LIN {X 0,Y 506.276,Z 611.91,A -85,B 0,C 180,E1 5620.333,E2 5620.333} C_VEL
LIN {X 0,Y 503.8,Z 611.91,A -85,B 0,C 180,E1 5621.794,E2 5621.794} C_VEL
LIN {X 0,Y 498.576,Z 611.91,A -85,B 0,C 180,E1 5623.986,E2 5623.986} C_VEL
LIN {X 0,Y 498.505,Z 611.91,A -85,B 0,C 180,E1 5624.239,E2 5624.239} C_VEL
LIN {X 0,Y 498.52,Z 611.91,A -85,B 0,C 180,E1 5630.373,E2 5630.373} C_VEL
LIN {X 0,Y 498.56,Z 611.91,A -85,B 0,C 180,E1 5636.864,E2 5636.864} C_VEL
LIN {X 0,Y 498.673,Z 612.016,A -85,B 0,C 180,E1 5638.544,E2 5638.544} C_VEL
LIN {X 0,Y 512.313,Z 645.051,A -85,B 0,C 180,E1 5639.998,E2 5639.998} C_VEL
LIN {X 0,Y 510.936,Z 684.615,A -85,B 0,C 180,E1 5640.995,E2 5640.995} C_VEL
LIN {X 0,Y 508.94,Z 720.292,A -85,B 0,C 180,E1 5642.602,E2 5642.602} C_VEL
LIN {X 0,Y 506.706,Z 753.658,A -85,B 0,C 180,E1 5644.799,E2 5644.799} C_VEL
LIN {X 0,Y 504.225,Z 785.399,A -85,B 0,C 180,E1 5647.723,E2 5647.723} C_VEL
LIN {X 0,Y 502.28,Z 810.959,A -85,B 0,C 180,E1 5650.895,E2 5650.895} C_VEL
LIN {X 0,Y 500.766,Z 834.651,A -85,B 0,C 180,E1 5654.902,E2 5654.902} C_VEL
LIN {X 0,Y 499.92,Z 850.471,A -85,B 0,C 180,E1 5658.647,E2 5658.647} C_VEL
LIN {X 0,Y 499.661,Z 861.793,A -85,B 0,C 180,E1 5662.601,E2 5662.601} C_VEL
LIN {X 0,Y 499.493,Z 868.21,A -85,B 0,C 180,E1 5666.524,E2 5666.524} C_VEL
LIN {X 0,Y 499.463,Z 870,A -85,B 0,C 180,E1 5670,E2 5670} C_VEL
LIN {X 0,Y 499.553,Z 867.136,A -85,B 0,C 180,E1 5674.346,E2 5674.346} C_VEL
LIN {X 0,Y 499.754,Z 858.648,A -85,B 0,C 180,E1 5678.713,E2 5678.713} C_VEL
LIN {X 0,Y 500.276,Z 843.684,A -85,B 0,C 180,E1 5683.12,E2 5683.12} C_VEL
LIN {X 0,Y 501.297,Z 824.914,A -85,B 0,C 180,E1 5686.9,E2 5686.9} C_VEL
LIN {X 0,Y 503.025,Z 800.805,A -85,B 0,C 180,E1 5690.481,E2 5690.481} C_VEL
LIN {X 0,Y 505.254,Z 771.947,A -85,B 0,C 180,E1 5693.626,E2 5693.626} C_VEL
LIN {X 0,Y 507.724,Z 739.674,A -85,B 0,C 180,E1 5696.213,E2 5696.213} C_VEL
LIN {X 0,Y 510.037,Z 703.559,A -85,B 0,C 180,E1 5698.236,E2 5698.236} C_VEL
LIN {X 0,Y 511.594,Z 668.352,A -85,B 0,C 180,E1 5699.506,E2 5699.506} C_VEL
LIN {X 0,Y 511.782,Z 643.626,A -85,B 0,C 180,E1 5700.064,E2 5700.064} C_VEL
LIN {X 0,Y 498.658,Z 611.91,A -85,B 0,C 180,E1 5701.494,E2 5701.494} C_VEL
LIN {X 0,Y 498.497,Z 611.91,A -85,B 0,C 180,E1 5707.852,E2 5707.852} C_VEL
LIN {X 0,Y 498.526,Z 611.91,A -85,B 0,C 180,E1 5714.309,E2 5714.309} C_VEL
LIN {X 0,Y 498.401,Z 611.91,A -85,B 0,C 180,E1 5720.367,E2 5720.367} C_VEL
LIN {X 0,Y 498.615,Z 611.91,A -85,B 0,C 180,E1 5726.873,E2 5726.873} C_VEL
LIN {X 0,Y 498.61,Z 611.91,A -85,B 0,C 180,E1 5732.909,E2 5732.909} C_VEL
LIN {X 0,Y 498.723,Z 611.91,A -85,B 0,C 180,E1 5738.64,E2 5738.64} C_VEL
LIN {X 0,Y 498.877,Z 611.91,A -85,B 0,C 180,E1 5744.153,E2 5744.153} C_VEL
LIN {X 0,Y 499.006,Z 611.91,A -85,B 0,C 180,E1 5749.515,E2 5749.515} C_VEL
LIN {X 0,Y 499.132,Z 611.91,A -85,B 0,C 180,E1 5754.782,E2 5754.782} C_VEL
LIN {X 0,Y 499.242,Z 611.91,A -85,B 0,C 180,E1 5760.003,E2 5760.003} C_VEL
LIN {X 0,Y 499.177,Z 611.91,A -85,B 0,C 180,E1 5765.224,E2 5765.224} C_VEL
LIN {X 0,Y 498.98,Z 611.91,A -85,B 0,C 180,E1 5770.492,E2 5770.492} C_VEL
LIN {X 0,Y 498.89,Z 611.91,A -85,B 0,C 180,E1 5775.854,E2 5775.854} C_VEL
LIN {X 0,Y 498.793,Z 611.91,A -85,B 0,C 180,E1 5781.364,E2 5781.364} C_VEL
LIN {X 0,Y 498.613,Z 611.91,A -85,B 0,C 180,E1 5787.098,E2 5787.098} C_VEL
LIN {X 0,Y 498.526,Z 611.91,A -85,B 0,C 180,E1 5793.141,E2 5793.141} C_VEL
LIN {X 0,Y 498.498,Z 611.91,A -85,B 0,C 180,E1 5799.632,E2 5799.632} C_VEL
LIN {X 0,Y 498.506,Z 611.91,A -85,B 0,C 180,E1 5805.689,E2 5805.689} C_VEL
LIN {X 0,Y 498.463,Z 611.91,A -85,B 0,C 180,E1 5812.163,E2 5812.163} C_VEL
LIN {X 0,Y 498.48,Z 611.91,A -85,B 0,C 180,E1 5818.263,E2 5818.263} C_VEL
LIN {X 0,Y 498.733,Z 611.91,A -85,B 0,C 180,E1 5824.849,E2 5824.849} C_VEL
LIN {X 0,Y 498.77,Z 611.91,A -85,B 0,C 180,E1 5830.494,E2 5830.494} C_VEL
LIN {X 0,Y 498.948,Z 611.91,A -85,B 0,C 180,E1 5836.18,E2 5836.18} C_VEL
LIN {X 0,Y 498.982,Z 611.91,A -85,B 0,C 180,E1 5841.274,E2 5841.274} C_VEL
LIN {X 0,Y 499.104,Z 611.91,A -85,B 0,C 180,E1 5846.522,E2 5846.522} C_VEL
LIN {X 0,Y 499.181,Z 611.91,A -85,B 0,C 180,E1 5851.738,E2 5851.738} C_VEL
LIN {X 0,Y 499.037,Z 611.91,A -85,B 0,C 180,E1 5856.97,E2 5856.97} C_VEL
LIN {X 0,Y 498.923,Z 611.91,A -85,B 0,C 180,E1 5862.264,E2 5862.264} C_VEL
LIN {X 0,Y 498.845,Z 611.91,A -85,B 0,C 180,E1 5867.669,E2 5867.669} C_VEL
LIN {X 0,Y 498.719,Z 611.91,A -85,B 0,C 180,E1 5873.245,E2 5873.245} C_VEL
LIN {X 0,Y 498.609,Z 611.91,A -85,B 0,C 180,E1 5879.068,E2 5879.068} C_VEL
LIN {X 0,Y 498.674,Z 611.91,A -85,B 0,C 180,E1 5885.231,E2 5885.231} C_VEL
LIN {X 0,Y 498.413,Z 611.91,A -85,B 0,C 180,E1 5891.936,E2 5891.936} C_VEL
LIN {X 0,Y 498.329,Z 611.91,A -85,B 0,C 180,E1 5898.053,E2 5898.053} C_VEL
LIN {X 0,Y 498.476,Z 611.91,A -85,B 0,C 180,E1 5904.751,E2 5904.751} C_VEL
LIN {X 0,Y 498.577,Z 611.91,A -85,B 0,C 180,E1 5910.928,E2 5910.928} C_VEL
LIN {X 0,Y 498.767,Z 611.91,A -85,B 0,C 180,E1 5916.755,E2 5916.755} C_VEL
LIN {X 0,Y 498.903,Z 611.91,A -85,B 0,C 180,E1 5922.331,E2 5922.331} C_VEL
LIN {X 0,Y 498.925,Z 611.91,A -85,B 0,C 180,E1 5929.506,E2 5929.506} C_VEL
LIN {X 0,Y 499.18,Z 611.91,A -85,B 0,C 180,E1 5934.776,E2 5934.776} C_VEL
LIN {X 0,Y 499.289,Z 611.91,A -85,B 0,C 180,E1 5939.997,E2 5939.997} C_VEL
LIN {X 0,Y 499.137,Z 611.91,A -85,B 0,C 180,E1 5945.218,E2 5945.218} C_VEL
LIN {X 0,Y 499.006,Z 611.91,A -85,B 0,C 180,E1 5950.485,E2 5950.485} C_VEL
LIN {X 0,Y 498.883,Z 611.91,A -85,B 0,C 180,E1 5955.847,E2 5955.847} C_VEL
LIN {X 0,Y 498.81,Z 611.91,A -85,B 0,C 180,E1 5961.357,E2 5961.357} C_VEL
LIN {X 0,Y 498.6,Z 611.91,A -85,B 0,C 180,E1 5967.092,E2 5967.092} C_VEL
LIN {X 0,Y 498.535,Z 611.91,A -85,B 0,C 180,E1 5973.133,E2 5973.133} C_VEL
LIN {X 0,Y 498.403,Z 611.91,A -85,B 0,C 180,E1 5979.632,E2 5979.632} C_VEL
LIN {X 0,Y 498.505,Z 611.91,A -85,B 0,C 180,E1 5984.239,E2 5984.239} C_VEL
LIN {X 0,Y 496.088,Z 611.91,A -85,B 0,C 180,E1 5985.715,E2 5985.715} C_VEL
LIN {X 0,Y 490.614,Z 611.91,A -85,B 0,C 180,E1 5988.184,E2 5988.184} C_VEL
LIN {X 0,Y 490.58,Z 611.91,A -85,B 0,C 180,E1 5994.099,E2 5994.099} C_VEL
LIN {X 0,Y 490.725,Z 611.91,A -85,B 0,C 180,E1 5997.959,E2 5997.959} C_VEL
LIN {X 0,Y 505.428,Z 648.806,A -85,B 0,C 180,E1 5999.626,E2 5999.626} C_VEL
LIN {X 0,Y 503.886,Z 686.608,A -85,B 0,C 180,E1 6000.634,E2 6000.634} C_VEL
LIN {X 0,Y 501.616,Z 724.072,A -85,B 0,C 180,E1 6002.411,E2 6002.411} C_VEL
LIN {X 0,Y 499.129,Z 756.38,A -85,B 0,C 180,E1 6004.647,E2 6004.647} C_VEL
LIN {X 0,Y 496.541,Z 788.376,A -85,B 0,C 180,E1 6007.713,E2 6007.713} C_VEL
LIN {X 0,Y 494.357,Z 814.607,A -85,B 0,C 180,E1 6011.146,E2 6011.146} C_VEL
LIN {X 0,Y 492.939,Z 835.779,A -85,B 0,C 180,E1 6014.886,E2 6014.886} C_VEL
LIN {X 0,Y 492.023,Z 851.964,A -85,B 0,C 180,E1 6018.912,E2 6018.912} C_VEL
LIN {X 0,Y 491.729,Z 862.787,A -85,B 0,C 180,E1 6022.925,E2 6022.925} C_VEL
LIN {X 0,Y 491.592,Z 868.213,A -85,B 0,C 180,E1 6026.468,E2 6026.468} C_VEL
LIN {X 0,Y 491.563,Z 870,A -85,B 0,C 180,E1 6030,E2 6030} C_VEL
LIN {X 0,Y 491.669,Z 867.131,A -85,B 0,C 180,E1 6034.415,E2 6034.415} C_VEL
LIN {X 0,Y 491.857,Z 858.643,A -85,B 0,C 180,E1 6038.854,E2 6038.854} C_VEL
LIN {X 0,Y 492.461,Z 843.681,A -85,B 0,C 180,E1 6043.332,E2 6043.332} C_VEL
LIN {X 0,Y 493.594,Z 824.909,A -85,B 0,C 180,E1 6047.172,E2 6047.172} C_VEL
LIN {X 0,Y 495.421,Z 801.229,A -85,B 0,C 180,E1 6050.74,E2 6050.74} C_VEL
LIN {X 0,Y 497.785,Z 772.507,A -85,B 0,C 180,E1 6053.924,E2 6053.924} C_VEL
LIN {X 0,Y 500.447,Z 740.735,A -85,B 0,C 180,E1 6056.534,E2 6056.534} C_VEL
LIN {X 0,Y 502.822,Z 705.679,A -85,B 0,C 180,E1 6058.556,E2 6058.556} C_VEL
LIN {X 0,Y 504.57,Z 671.257,A -85,B 0,C 180,E1 6059.87,E2 6059.87} C_VEL
LIN {X 0,Y 504.936,Z 645.854,A -85,B 0,C 180,E1 6060.466,E2 6060.466} C_VEL
LIN {X 0,Y 490.719,Z 611.91,A -85,B 0,C 180,E1 6062.086,E2 6062.086} C_VEL
LIN {X 0,Y 490.57,Z 611.91,A -85,B 0,C 180,E1 6068.117,E2 6068.117} C_VEL
LIN {X 0,Y 490.648,Z 611.91,A -85,B 0,C 180,E1 6072.756,E2 6072.756} C_VEL
LIN {X 0,Y 490.538,Z 611.91,A -85,B 0,C 180,E1 6077.797,E2 6077.797} C_VEL
LIN {X 0,Y 490.553,Z 611.91,A -85,B 0,C 180,E1 6084.102,E2 6084.102} C_VEL
LIN {X 0,Y 490.666,Z 611.91,A -85,B 0,C 180,E1 6090.42,E2 6090.42} C_VEL
LIN {X 0,Y 490.743,Z 611.91,A -85,B 0,C 180,E1 6096.359,E2 6096.359} C_VEL
LIN {X 0,Y 490.906,Z 611.91,A -85,B 0,C 180,E1 6102.96,E2 6102.96} C_VEL
LIN {X 0,Y 491.088,Z 611.91,A -85,B 0,C 180,E1 6109.344,E2 6109.344} C_VEL
LIN {X 0,Y 491.216,Z 611.91,A -85,B 0,C 180,E1 6114.698,E2 6114.698} C_VEL
LIN {X 0,Y 491.342,Z 611.91,A -85,B 0,C 180,E1 6120.003,E2 6120.003} C_VEL
LIN {X 0,Y 491.265,Z 611.91,A -85,B 0,C 180,E1 6125.308,E2 6125.308} C_VEL
LIN {X 0,Y 491.069,Z 611.91,A -85,B 0,C 180,E1 6130.663,E2 6130.663} C_VEL
LIN {X 0,Y 490.926,Z 611.91,A -85,B 0,C 180,E1 6137.047,E2 6137.047} C_VEL
LIN {X 0,Y 490.812,Z 611.91,A -85,B 0,C 180,E1 6143.645,E2 6143.645} C_VEL
LIN {X 0,Y 490.587,Z 611.91,A -85,B 0,C 180,E1 6150.215,E2 6150.215} C_VEL
LIN {X 0,Y 490.57,Z 611.91,A -85,B 0,C 180,E1 6156.636,E2 6156.636} C_VEL
LIN {X 0,Y 490.572,Z 611.91,A -85,B 0,C 180,E1 6162.767,E2 6162.767} C_VEL
LIN {X 0,Y 490.592,Z 611.91,A -85,B 0,C 180,E1 6167.792,E2 6167.792} C_VEL
LIN {X 0,Y 490.532,Z 611.91,A -85,B 0,C 180,E1 6174.095,E2 6174.095} C_VEL
LIN {X 0,Y 490.599,Z 611.91,A -85,B 0,C 180,E1 6180.411,E2 6180.411} C_VEL
LIN {X 0,Y 490.816,Z 611.91,A -85,B 0,C 180,E1 6186.358,E2 6186.358} C_VEL
LIN {X 0,Y 490.924,Z 611.91,A -85,B 0,C 180,E1 6192.957,E2 6192.957} C_VEL
LIN {X 0,Y 491.074,Z 611.91,A -85,B 0,C 180,E1 6199.34,E2 6199.34} C_VEL
LIN {X 0,Y 491.241,Z 611.91,A -85,B 0,C 180,E1 6204.695,E2 6204.695} C_VEL
LIN {X 0,Y 491.348,Z 611.91,A -85,B 0,C 180,E1 6210,E2 6210} C_VEL
LIN {X 0,Y 491.207,Z 611.91,A -85,B 0,C 180,E1 6215.306,E2 6215.306} C_VEL
LIN {X 0,Y 491.067,Z 611.91,A -85,B 0,C 180,E1 6220.661,E2 6220.661} C_VEL
LIN {X 0,Y 490.929,Z 611.91,A -85,B 0,C 180,E1 6227.045,E2 6227.045} C_VEL
LIN {X 0,Y 490.786,Z 611.91,A -85,B 0,C 180,E1 6232.255,E2 6232.255} C_VEL
LIN {X 0,Y 490.677,Z 611.91,A -85,B 0,C 180,E1 6237.571,E2 6237.571} C_VEL
LIN {X 0,Y 490.731,Z 611.91,A -85,B 0,C 180,E1 6243.735,E2 6243.735} C_VEL
LIN {X 0,Y 490.552,Z 611.91,A -85,B 0,C 180,E1 6250.402,E2 6250.402} C_VEL
LIN {X 0,Y 490.423,Z 611.91,A -85,B 0,C 180,E1 6257.217,E2 6257.217} C_VEL
LIN {X 0,Y 490.447,Z 611.91,A -85,B 0,C 180,E1 6263.383,E2 6263.383} C_VEL
LIN {X 0,Y 490.613,Z 611.91,A -85,B 0,C 180,E1 6268.354,E2 6268.354} C_VEL
LIN {X 0,Y 490.756,Z 611.91,A -85,B 0,C 180,E1 6274.408,E2 6274.408} C_VEL
LIN {X 0,Y 490.998,Z 611.91,A -85,B 0,C 180,E1 6280.169,E2 6280.169} C_VEL
LIN {X 0,Y 490.812,Z 611.91,A -85,B 0,C 180,E1 6285.71,E2 6285.71} C_VEL
LIN {X 0,Y 491.056,Z 611.91,A -85,B 0,C 180,E1 6291.425,E2 6291.425} C_VEL
LIN {X 0,Y 491.243,Z 611.91,A -85,B 0,C 180,E1 6296.463,E2 6296.463} C_VEL
LIN {X 0,Y 491.272,Z 611.91,A -85,B 0,C 180,E1 6301.763,E2 6301.763} C_VEL
LIN {X 0,Y 491.124,Z 611.91,A -85,B 0,C 180,E1 6307.08,E2 6307.08} C_VEL
LIN {X 0,Y 491.02,Z 611.91,A -85,B 0,C 180,E1 6312.461,E2 6312.461} C_VEL
LIN {X 0,Y 490.926,Z 611.91,A -85,B 0,C 180,E1 6317.959,E2 6317.959} C_VEL
LIN {X 0,Y 490.81,Z 611.91,A -85,B 0,C 180,E1 6323.638,E2 6323.638} C_VEL
LIN {X 0,Y 490.593,Z 611.91,A -85,B 0,C 180,E1 6330.217,E2 6330.217} C_VEL
LIN {X 0,Y 490.527,Z 611.91,A -85,B 0,C 180,E1 6335.9,E2 6335.9} C_VEL
LIN {X 0,Y 490.541,Z 611.91,A -85,B 0,C 180,E1 6342.204,E2 6342.204} C_VEL
LIN {X 0,Y 490.614,Z 611.91,A -85,B 0,C 180,E1 6348.184,E2 6348.184} C_VEL
LIN {X 0,Y 486.597,Z 611.91,A -85,B 0,C 180,E1 6350.167,E2 6350.167} C_VEL
LIN {X 0,Y 482.62,Z 611.91,A -85,B 0,C 180,E1 6352.182,E2 6352.182} C_VEL
LIN {X 0,Y 482.789,Z 611.91,A -85,B 0,C 180,E1 6357.349,E2 6357.349} C_VEL
LIN {X 0,Y 498.578,Z 650.929,A -85,B 0,C 180,E1 6359.211,E2 6359.211} C_VEL
LIN {X 0,Y 496.886,Z 687.431,A -85,B 0,C 180,E1 6360.225,E2 6360.225} C_VEL
LIN {X 0,Y 494.448,Z 724.843,A -85,B 0,C 180,E1 6362.038,E2 6362.038} C_VEL
LIN {X 0,Y 491.718,Z 757.47,A -85,B 0,C 180,E1 6364.358,E2 6364.358} C_VEL
LIN {X 0,Y 488.948,Z 789.177,A -85,B 0,C 180,E1 6367.468,E2 6367.468} C_VEL
LIN {X 0,Y 486.509,Z 816.896,A -85,B 0,C 180,E1 6371.217,E2 6371.217} C_VEL
LIN {X 0,Y 485.077,Z 836.82,A -85,B 0,C 180,E1 6374.87,E2 6374.87} C_VEL
LIN {X 0,Y 484.122,Z 853.457,A -85,B 0,C 180,E1 6379.185,E2 6379.185} C_VEL
LIN {X 0,Y 483.847,Z 862.789,A -85,B 0,C 180,E1 6382.81,E2 6382.81} C_VEL
LIN {X 0,Y 483.71,Z 868.216,A -85,B 0,C 180,E1 6386.411,E2 6386.411} C_VEL
LIN {X 0,Y 483.671,Z 870,A -85,B 0,C 180,E1 6390,E2 6390} C_VEL
LIN {X 0,Y 483.78,Z 867.127,A -85,B 0,C 180,E1 6394.487,E2 6394.487} C_VEL
LIN {X 0,Y 483.981,Z 858.637,A -85,B 0,C 180,E1 6398.999,E2 6398.999} C_VEL
LIN {X 0,Y 484.64,Z 843.678,A -85,B 0,C 180,E1 6403.551,E2 6403.551} C_VEL
LIN {X 0,Y 485.866,Z 824.842,A -85,B 0,C 180,E1 6407.454,E2 6407.454} C_VEL
LIN {X 0,Y 487.843,Z 800.722,A -85,B 0,C 180,E1 6411.115,E2 6411.115} C_VEL
LIN {X 0,Y 490.366,Z 772.74,A -85,B 0,C 180,E1 6414.261,E2 6414.261} C_VEL
LIN {X 0,Y 493.269,Z 740.307,A -85,B 0,C 180,E1 6416.965,E2 6416.965} C_VEL
LIN {X 0,Y 495.945,Z 704.265,A -85,B 0,C 180,E1 6419.052,E2 6419.052} C_VEL
LIN {X 0,Y 497.776,Z 669.559,A -85,B 0,C 180,E1 6420.362,E2 6420.362} C_VEL
LIN {X 0,Y 498.125,Z 648.288,A -85,B 0,C 180,E1 6420.873,E2 6420.873} C_VEL
LIN {X 0,Y 482.776,Z 611.91,A -85,B 0,C 180,E1 6422.721,E2 6422.721} C_VEL
LIN {X 0,Y 482.644,Z 611.91,A -85,B 0,C 180,E1 6428.859,E2 6428.859} C_VEL
LIN {X 0,Y 482.646,Z 611.91,A -85,B 0,C 180,E1 6433.828,E2 6433.828} C_VEL
LIN {X 0,Y 482.554,Z 611.91,A -85,B 0,C 180,E1 6438.853,E2 6438.853} C_VEL
LIN {X 0,Y 482.621,Z 611.91,A -85,B 0,C 180,E1 6444.653,E2 6444.653} C_VEL
LIN {X 0,Y 482.774,Z 611.91,A -85,B 0,C 180,E1 6449.887,E2 6449.887} C_VEL
LIN {X 0,Y 482.789,Z 611.91,A -85,B 0,C 180,E1 6455.945,E2 6455.945} C_VEL
LIN {X 0,Y 482.949,Z 611.91,A -85,B 0,C 180,E1 6461.734,E2 6461.734} C_VEL
LIN {X 0,Y 483.094,Z 611.91,A -85,B 0,C 180,E1 6467.331,E2 6467.331} C_VEL
LIN {X 0,Y 483.233,Z 611.91,A -85,B 0,C 180,E1 6472.804,E2 6472.804} C_VEL
LIN {X 0,Y 483.386,Z 611.91,A -85,B 0,C 180,E1 6478.208,E2 6478.208} C_VEL
LIN {X 0,Y 483.343,Z 611.91,A -85,B 0,C 180,E1 6483.595,E2 6483.595} C_VEL
LIN {X 0,Y 483.163,Z 611.91,A -85,B 0,C 180,E1 6489.017,E2 6489.017} C_VEL
LIN {X 0,Y 483.058,Z 611.91,A -85,B 0,C 180,E1 6494.524,E2 6494.524} C_VEL
LIN {X 0,Y 482.955,Z 611.91,A -85,B 0,C 180,E1 6500.175,E2 6500.175} C_VEL
LIN {X 0,Y 482.824,Z 611.91,A -85,B 0,C 180,E1 6506.044,E2 6506.044} C_VEL
LIN {X 0,Y 482.658,Z 611.91,A -85,B 0,C 180,E1 6512.229,E2 6512.229} C_VEL
LIN {X 0,Y 482.659,Z 611.91,A -85,B 0,C 180,E1 6518.859,E2 6518.859} C_VEL
LIN {X 0,Y 482.604,Z 611.91,A -85,B 0,C 180,E1 6523.816,E2 6523.816} C_VEL
LIN {X 0,Y 482.627,Z 611.91,A -85,B 0,C 180,E1 6528.845,E2 6528.845} C_VEL
LIN {X 0,Y 482.578,Z 611.91,A -85,B 0,C 180,E1 6534.662,E2 6534.662} C_VEL
LIN {X 0,Y 482.687,Z 611.91,A -85,B 0,C 180,E1 6539.876,E2 6539.876} C_VEL
LIN {X 0,Y 482.857,Z 611.91,A -85,B 0,C 180,E1 6545.944,E2 6545.944} C_VEL
LIN {X 0,Y 482.969,Z 611.91,A -85,B 0,C 180,E1 6551.73,E2 6551.73} C_VEL
LIN {X 0,Y 483.094,Z 611.91,A -85,B 0,C 180,E1 6557.327,E2 6557.327} C_VEL
LIN {X 0,Y 483.292,Z 611.91,A -85,B 0,C 180,E1 6562.801,E2 6562.801} C_VEL
LIN {X 0,Y 483.561,Z 611.91,A -85,B 0,C 180,E1 6568.206,E2 6568.206} C_VEL
LIN {X 0,Y 483.428,Z 611.91,A -85,B 0,C 180,E1 6573.591,E2 6573.591} C_VEL
LIN {X 0,Y 483.214,Z 611.91,A -85,B 0,C 180,E1 6579.013,E2 6579.013} C_VEL
LIN {X 0,Y 483.096,Z 611.91,A -85,B 0,C 180,E1 6584.52,E2 6584.52} C_VEL
LIN {X 0,Y 482.966,Z 611.91,A -85,B 0,C 180,E1 6590.172,E2 6590.172} C_VEL
LIN {X 0,Y 482.821,Z 611.91,A -85,B 0,C 180,E1 6596.041,E2 6596.041} C_VEL
LIN {X 0,Y 482.803,Z 611.91,A -85,B 0,C 180,E1 6602.216,E2 6602.216} C_VEL
LIN {X 0,Y 482.696,Z 611.91,A -85,B 0,C 180,E1 6608.354,E2 6608.354} C_VEL
LIN {X 0,Y 482.478,Z 611.91,A -85,B 0,C 180,E1 6613.798,E2 6613.798} C_VEL
LIN {X 0,Y 482.495,Z 611.91,A -85,B 0,C 180,E1 6618.861,E2 6618.861} C_VEL
LIN {X 0,Y 482.536,Z 611.91,A -85,B 0,C 180,E1 6624.667,E2 6624.667} C_VEL
LIN {X 0,Y 482.689,Z 611.91,A -85,B 0,C 180,E1 6629.874,E2 6629.874} C_VEL
LIN {X 0,Y 482.872,Z 611.91,A -85,B 0,C 180,E1 6635.942,E2 6635.942} C_VEL
LIN {X 0,Y 483.053,Z 611.91,A -85,B 0,C 180,E1 6641.731,E2 6641.731} C_VEL
LIN {X 0,Y 482.935,Z 611.91,A -85,B 0,C 180,E1 6647.32,E2 6647.32} C_VEL
LIN {X 0,Y 483.315,Z 611.91,A -85,B 0,C 180,E1 6652.799,E2 6652.799} C_VEL
LIN {X 0,Y 483.587,Z 611.91,A -85,B 0,C 180,E1 6658.203,E2 6658.203} C_VEL
LIN {X 0,Y 483.478,Z 611.91,A -85,B 0,C 180,E1 6663.587,E2 6663.587} C_VEL
LIN {X 0,Y 483.229,Z 611.91,A -85,B 0,C 180,E1 6669.009,E2 6669.009} C_VEL
LIN {X 0,Y 483.089,Z 611.91,A -85,B 0,C 180,E1 6674.517,E2 6674.517} C_VEL
LIN {X 0,Y 482.974,Z 611.91,A -85,B 0,C 180,E1 6680.167,E2 6680.167} C_VEL
LIN {X 0,Y 482.816,Z 611.91,A -85,B 0,C 180,E1 6686.037,E2 6686.037} C_VEL
LIN {X 0,Y 482.696,Z 611.91,A -85,B 0,C 180,E1 6692.219,E2 6692.219} C_VEL
LIN {X 0,Y 482.57,Z 611.91,A -85,B 0,C 180,E1 6698.86,E2 6698.86} C_VEL
LIN {X 0,Y 482.604,Z 611.91,A -85,B 0,C 180,E1 6703.816,E2 6703.816} C_VEL
LIN {X 0,Y 482.685,Z 611.91,A -85,B 0,C 180,E1 6708.827,E2 6708.827} C_VEL
LIN {X 0,Y 482.62,Z 611.91,A -85,B 0,C 180,E1 6712.182,E2 6712.182} C_VEL
LIN {X 0,Y 481.331,Z 611.91,A -85,B 0,C 180,E1 6713.209,E2 6713.209} C_VEL
LIN {X 0,Y 474.852,Z 611.91,A -85,B 0,C 180,E1 6716.009,E2 6716.009} C_VEL
LIN {X 0,Y 474.786,Z 611.91,A -85,B 0,C 180,E1 6716.275,E2 6716.275} C_VEL
LIN {X 0,Y 474.851,Z 611.91,A -85,B 0,C 180,E1 6716.753,E2 6716.753} C_VEL
LIN {X 0,Y 491.664,Z 651.449,A -85,B 0,C 180,E1 6718.746,E2 6718.746} C_VEL
LIN {X 0,Y 489.989,Z 687.523,A -85,B 0,C 180,E1 6719.778,E2 6719.778} C_VEL
LIN {X 0,Y 487.394,Z 724.606,A -85,B 0,C 180,E1 6721.597,E2 6721.597} C_VEL
LIN {X 0,Y 484.463,Z 757.388,A -85,B 0,C 180,E1 6723.96,E2 6723.96} C_VEL
LIN {X 0,Y 481.456,Z 788.936,A -85,B 0,C 180,E1 6727.098,E2 6727.098} C_VEL
LIN {X 0,Y 478.876,Z 816.312,A -85,B 0,C 180,E1 6730.851,E2 6730.851} C_VEL
LIN {X 0,Y 477.215,Z 837.581,A -85,B 0,C 180,E1 6734.826,E2 6734.826} C_VEL
LIN {X 0,Y 476.266,Z 853.453,A -85,B 0,C 180,E1 6739.004,E2 6739.004} C_VEL
LIN {X 0,Y 475.963,Z 862.789,A -85,B 0,C 180,E1 6742.69,E2 6742.69} C_VEL
LIN {X 0,Y 475.811,Z 868.218,A -85,B 0,C 180,E1 6746.351,E2 6746.351} C_VEL
LIN {X 0,Y 475.771,Z 870,A -85,B 0,C 180,E1 6750,E2 6750} C_VEL
LIN {X 0,Y 475.834,Z 868.218,A -85,B 0,C 180,E1 6753.649,E2 6753.649} C_VEL
LIN {X 0,Y 476.084,Z 860.768,A -85,B 0,C 180,E1 6758.228,E2 6758.228} C_VEL
LIN {X 0,Y 476.537,Z 848.934,A -85,B 0,C 180,E1 6762.384,E2 6762.384} C_VEL
LIN {X 0,Y 477.717,Z 829.729,A -85,B 0,C 180,E1 6766.795,E2 6766.795} C_VEL
LIN {X 0,Y 479.677,Z 807.486,A -85,B 0,C 180,E1 6770.49,E2 6770.49} C_VEL
LIN {X 0,Y 482.444,Z 778.309,A -85,B 0,C 180,E1 6774.078,E2 6774.078} C_VEL
LIN {X 0,Y 485.532,Z 746.058,A -85,B 0,C 180,E1 6776.945,E2 6776.945} C_VEL
LIN {X 0,Y 488.326,Z 712.284,A -85,B 0,C 180,E1 6779.104,E2 6779.104} C_VEL
LIN {X 0,Y 490.714,Z 673.385,A -85,B 0,C 180,E1 6780.711,E2 6780.711} C_VEL
LIN {X 0,Y 491.152,Z 650.167,A -85,B 0,C 180,E1 6781.317,E2 6781.317} C_VEL
LIN {X 0,Y 474.827,Z 611.91,A -85,B 0,C 180,E1 6783.251,E2 6783.251} C_VEL
LIN {X 0,Y 474.66,Z 611.91,A -85,B 0,C 180,E1 6790.053,E2 6790.053} C_VEL
LIN {X 0,Y 474.628,Z 611.91,A -85,B 0,C 180,E1 6795.436,E2 6795.436} C_VEL
LIN {X 0,Y 474.577,Z 611.91,A -85,B 0,C 180,E1 6800.359,E2 6800.359} C_VEL
LIN {X 0,Y 474.734,Z 611.91,A -85,B 0,C 180,E1 6806.018,E2 6806.018} C_VEL
LIN {X 0,Y 474.82,Z 611.91,A -85,B 0,C 180,E1 6811.43,E2 6811.43} C_VEL
LIN {X 0,Y 474.917,Z 611.91,A -85,B 0,C 180,E1 6817.598,E2 6817.598} C_VEL
LIN {X 0,Y 475.072,Z 611.91,A -85,B 0,C 180,E1 6823.336,E2 6823.336} C_VEL
LIN {X 0,Y 475.231,Z 611.91,A -85,B 0,C 180,E1 6828.984,E2 6828.984} C_VEL
LIN {X 0,Y 475.4,Z 611.91,A -85,B 0,C 180,E1 6834.521,E2 6834.521} C_VEL
LIN {X 0,Y 475.541,Z 611.91,A -85,B 0,C 180,E1 6840.003,E2 6840.003} C_VEL
LIN {X 0,Y 475.45,Z 611.91,A -85,B 0,C 180,E1 6845.485,E2 6845.485} C_VEL
LIN {X 0,Y 475.214,Z 611.91,A -85,B 0,C 180,E1 6851.024,E2 6851.024} C_VEL
LIN {X 0,Y 475.069,Z 611.91,A -85,B 0,C 180,E1 6857.039,E2 6857.039} C_VEL
LIN {X 0,Y 474.978,Z 611.91,A -85,B 0,C 180,E1 6862.492,E2 6862.492} C_VEL
LIN {X 0,Y 474.763,Z 611.91,A -85,B 0,C 180,E1 6868.581,E2 6868.581} C_VEL
LIN {X 0,Y 474.713,Z 611.91,A -85,B 0,C 180,E1 6875.039,E2 6875.039} C_VEL
LIN {X 0,Y 474.647,Z 611.91,A -85,B 0,C 180,E1 6880.043,E2 6880.043} C_VEL
LIN {X 0,Y 474.629,Z 611.91,A -85,B 0,C 180,E1 6885.429,E2 6885.429} C_VEL
LIN {X 0,Y 474.634,Z 611.91,A -85,B 0,C 180,E1 6890.358,E2 6890.358} C_VEL
LIN {X 0,Y 474.639,Z 611.91,A -85,B 0,C 180,E1 6896.037,E2 6896.037} C_VEL
LIN {X 0,Y 474.775,Z 611.91,A -85,B 0,C 180,E1 6901.422,E2 6901.422} C_VEL
LIN {X 0,Y 474.981,Z 611.91,A -85,B 0,C 180,E1 6907.582,E2 6907.582} C_VEL
LIN {X 0,Y 475.088,Z 611.91,A -85,B 0,C 180,E1 6913.332,E2 6913.332} C_VEL
LIN {X 0,Y 475.22,Z 611.91,A -85,B 0,C 180,E1 6918.979,E2 6918.979} C_VEL
LIN {X 0,Y 475.429,Z 611.91,A -85,B 0,C 180,E1 6924.518,E2 6924.518} C_VEL
LIN {X 0,Y 475.547,Z 611.91,A -85,B 0,C 180,E1 6930,E2 6930} C_VEL
LIN {X 0,Y 475.393,Z 611.91,A -85,B 0,C 180,E1 6935.483,E2 6935.483} C_VEL
LIN {X 0,Y 475.215,Z 611.91,A -85,B 0,C 180,E1 6941.021,E2 6941.021} C_VEL
LIN {X 0,Y 475.059,Z 611.91,A -85,B 0,C 180,E1 6947.031,E2 6947.031} C_VEL
LIN {X 0,Y 474.972,Z 611.91,A -85,B 0,C 180,E1 6952.49,E2 6952.49} C_VEL
LIN {X 0,Y 474.795,Z 611.91,A -85,B 0,C 180,E1 6958.576,E2 6958.576} C_VEL
LIN {X 0,Y 474.832,Z 611.91,A -85,B 0,C 180,E1 6965.026,E2 6965.026} C_VEL
LIN {X 0,Y 474.63,Z 611.91,A -85,B 0,C 180,E1 6970.038,E2 6970.038} C_VEL
LIN {X 0,Y 474.478,Z 611.91,A -85,B 0,C 180,E1 6975.408,E2 6975.408} C_VEL
LIN {X 0,Y 474.534,Z 611.91,A -85,B 0,C 180,E1 6980.346,E2 6980.346} C_VEL
LIN {X 0,Y 474.621,Z 611.91,A -85,B 0,C 180,E1 6986.038,E2 6986.038} C_VEL
LIN {X 0,Y 474.774,Z 611.91,A -85,B 0,C 180,E1 6991.42,E2 6991.42} C_VEL
LIN {X 0,Y 475.029,Z 611.91,A -85,B 0,C 180,E1 6997.565,E2 6997.565} C_VEL
LIN {X 0,Y 475.073,Z 611.91,A -85,B 0,C 180,E1 7003.329,E2 7003.329} C_VEL
LIN {X 0,Y 475.144,Z 611.91,A -85,B 0,C 180,E1 7008.975,E2 7008.975} C_VEL
LIN {X 0,Y 475.453,Z 611.91,A -85,B 0,C 180,E1 7014.515,E2 7014.515} C_VEL
LIN {X 0,Y 475.614,Z 611.91,A -85,B 0,C 180,E1 7019.997,E2 7019.997} C_VEL
LIN {X 0,Y 475.403,Z 611.91,A -85,B 0,C 180,E1 7025.479,E2 7025.479} C_VEL
LIN {X 0,Y 475.231,Z 611.91,A -85,B 0,C 180,E1 7031.016,E2 7031.016} C_VEL
LIN {X 0,Y 475.055,Z 611.91,A -85,B 0,C 180,E1 7037.034,E2 7037.034} C_VEL
LIN {X 0,Y 475,Z 611.91,A -85,B 0,C 180,E1 7042.484,E2 7042.484} C_VEL
LIN {X 0,Y 474.76,Z 611.91,A -85,B 0,C 180,E1 7048.574,E2 7048.574} C_VEL
LIN {X 0,Y 474.677,Z 611.91,A -85,B 0,C 180,E1 7055.034,E2 7055.034} C_VEL
LIN {X 0,Y 474.574,Z 611.91,A -85,B 0,C 180,E1 7062.058,E2 7062.058} C_VEL
LIN {X 0,Y 474.681,Z 611.91,A -85,B 0,C 180,E1 7067.947,E2 7067.947} C_VEL
LIN {X 0,Y 474.723,Z 611.91,A -85,B 0,C 180,E1 7074.965,E2 7074.965} C_VEL
LIN {X 0,Y 474.786,Z 611.91,A -85,B 0,C 180,E1 7076.275,E2 7076.275} C_VEL
LIN {X 0,Y 475.818,Z 614.619,A -85,B 0,C 180,E1 7076.84,E2 7076.84} C_VEL
LIN {X 0,Y 478.441,Z 624.168,A -85,B 0,C 180,E1 7077.274,E2 7077.274} C_VEL
LIN {X 0,Y 481.023,Z 644.057,A -85,B 0,C 180,E1 7077.823,E2 7077.823} C_VEL
LIN {X 0,Y 484.867,Z 655.755,A -85,B 0,C 180,E1 7078.353,E2 7078.353} C_VEL
LIN {X 0,Y 482.753,Z 693.603,A -85,B 0,C 180,E1 7079.568,E2 7079.568} C_VEL
LIN {X 0,Y 480.033,Z 728.244,A -85,B 0,C 180,E1 7081.378,E2 7081.378} C_VEL
LIN {X 0,Y 476.749,Z 761.976,A -85,B 0,C 180,E1 7083.959,E2 7083.959} C_VEL
LIN {X 0,Y 473.807,Z 790.609,A -85,B 0,C 180,E1 7086.955,E2 7086.955} C_VEL
LIN {X 0,Y 471.11,Z 817.577,A -85,B 0,C 180,E1 7090.767,E2 7090.767} C_VEL
LIN {X 0,Y 469.342,Z 838.371,A -85,B 0,C 180,E1 7094.805,E2 7094.805} C_VEL
LIN {X 0,Y 468.397,Z 853.272,A -85,B 0,C 180,E1 7098.817,E2 7098.817} C_VEL
LIN {X 0,Y 468.093,Z 862.743,A -85,B 0,C 180,E1 7102.566,E2 7102.566} C_VEL
LIN {X 0,Y 467.913,Z 868.218,A -85,B 0,C 180,E1 7106.29,E2 7106.29} C_VEL
LIN {X 0,Y 467.879,Z 870,A -85,B 0,C 180,E1 7110,E2 7110} C_VEL
LIN {X 0,Y 467.935,Z 868.218,A -85,B 0,C 180,E1 7113.71,E2 7113.71} C_VEL
LIN {X 0,Y 468.195,Z 860.695,A -85,B 0,C 180,E1 7118.367,E2 7118.367} C_VEL
LIN {X 0,Y 468.691,Z 848.697,A -85,B 0,C 180,E1 7122.595,E2 7122.595} C_VEL
LIN {X 0,Y 470.023,Z 829.588,A -85,B 0,C 180,E1 7127.058,E2 7127.058} C_VEL
LIN {X 0,Y 472.128,Z 806.506,A -85,B 0,C 180,E1 7130.94,E2 7130.94} C_VEL
LIN {X 0,Y 475.063,Z 778.07,A -85,B 0,C 180,E1 7134.476,E2 7134.476} C_VEL
LIN {X 0,Y 478.394,Z 745.617,A -85,B 0,C 180,E1 7137.397,E2 7137.397} C_VEL
LIN {X 0,Y 481.365,Z 712.048,A -85,B 0,C 180,E1 7139.566,E2 7139.566} C_VEL
LIN {X 0,Y 483.87,Z 673.96,A -85,B 0,C 180,E1 7141.163,E2 7141.163} C_VEL
LIN {X 0,Y 484.197,Z 652.012,A -85,B 0,C 180,E1 7141.775,E2 7141.775} C_VEL
LIN {X 0,Y 466.845,Z 611.91,A -85,B 0,C 180,E1 7143.911,E2 7143.911} C_VEL
LIN {X 0,Y 466.724,Z 611.91,A -85,B 0,C 180,E1 7150.451,E2 7150.451} C_VEL
LIN {X 0,Y 466.705,Z 611.91,A -85,B 0,C 180,E1 7157.064,E2 7157.064} C_VEL
LIN {X 0,Y 466.735,Z 611.91,A -85,B 0,C 180,E1 7164.192,E2 7164.192} C_VEL
LIN {X 0,Y 466.844,Z 611.91,A -85,B 0,C 180,E1 7168.746,E2 7168.746} C_VEL
LIN {X 0,Y 466.952,Z 611.91,A -85,B 0,C 180,E1 7175.214,E2 7175.214} C_VEL
LIN {X 0,Y 467.067,Z 611.91,A -85,B 0,C 180,E1 7181.09,E2 7181.09} C_VEL
LIN {X 0,Y 467.247,Z 611.91,A -85,B 0,C 180,E1 7186.894,E2 7186.894} C_VEL
LIN {X 0,Y 467.405,Z 611.91,A -85,B 0,C 180,E1 7192.559,E2 7192.559} C_VEL
LIN {X 0,Y 467.58,Z 611.91,A -85,B 0,C 180,E1 7198.148,E2 7198.148} C_VEL
LIN {X 0,Y 467.529,Z 611.91,A -85,B 0,C 180,E1 7203.717,E2 7203.717} C_VEL
LIN {X 0,Y 467.34,Z 611.91,A -85,B 0,C 180,E1 7209.325,E2 7209.325} C_VEL
LIN {X 0,Y 467.194,Z 611.91,A -85,B 0,C 180,E1 7215.029,E2 7215.029} C_VEL
LIN {X 0,Y 467.082,Z 611.91,A -85,B 0,C 180,E1 7220.892,E2 7220.892} C_VEL
LIN {X 0,Y 466.883,Z 611.91,A -85,B 0,C 180,E1 7227.004,E2 7227.004} C_VEL
LIN {X 0,Y 466.76,Z 611.91,A -85,B 0,C 180,E1 7233.468,E2 7233.468} C_VEL
LIN {X 0,Y 466.707,Z 611.91,A -85,B 0,C 180,E1 7240.455,E2 7240.455} C_VEL
LIN {X 0,Y 466.744,Z 611.91,A -85,B 0,C 180,E1 7247.062,E2 7247.062} C_VEL
LIN {X 0,Y 466.674,Z 611.91,A -85,B 0,C 180,E1 7251.944,E2 7251.944} C_VEL
LIN {X 0,Y 466.752,Z 611.91,A -85,B 0,C 180,E1 7258.734,E2 7258.734} C_VEL
LIN {X 0,Y 467.012,Z 611.91,A -85,B 0,C 180,E1 7265.201,E2 7265.201} C_VEL
LIN {X 0,Y 467.093,Z 611.91,A -85,B 0,C 180,E1 7271.086,E2 7271.086} C_VEL
LIN {X 0,Y 467.244,Z 611.91,A -85,B 0,C 180,E1 7276.89,E2 7276.89} C_VEL
LIN {X 0,Y 467.444,Z 611.91,A -85,B 0,C 180,E1 7282.556,E2 7282.556} C_VEL
LIN {X 0,Y 467.752,Z 611.91,A -85,B 0,C 180,E1 7288.145,E2 7288.145} C_VEL
LIN {X 0,Y 467.602,Z 611.91,A -85,B 0,C 180,E1 7293.713,E2 7293.713} C_VEL
LIN {X 0,Y 467.378,Z 611.91,A -85,B 0,C 180,E1 7299.321,E2 7299.321} C_VEL
LIN {X 0,Y 467.22,Z 611.91,A -85,B 0,C 180,E1 7305.025,E2 7305.025} C_VEL
LIN {X 0,Y 467.086,Z 611.91,A -85,B 0,C 180,E1 7310.889,E2 7310.889} C_VEL
LIN {X 0,Y 466.892,Z 611.91,A -85,B 0,C 180,E1 7317,E2 7317} C_VEL
LIN {X 0,Y 466.886,Z 611.91,A -85,B 0,C 180,E1 7323.456,E2 7323.456} C_VEL
LIN {X 0,Y 466.726,Z 611.91,A -85,B 0,C 180,E1 7328.869,E2 7328.869} C_VEL
LIN {X 0,Y 466.572,Z 611.91,A -85,B 0,C 180,E1 7335.554,E2 7335.554} C_VEL
LIN {X 0,Y 466.607,Z 611.91,A -85,B 0,C 180,E1 7341.935,E2 7341.935} C_VEL
LIN {X 0,Y 466.751,Z 611.91,A -85,B 0,C 180,E1 7348.732,E2 7348.732} C_VEL
LIN {X 0,Y 467.016,Z 611.91,A -85,B 0,C 180,E1 7355.197,E2 7355.197} C_VEL
LIN {X 0,Y 467.188,Z 611.91,A -85,B 0,C 180,E1 7361.087,E2 7361.087} C_VEL
LIN {X 0,Y 467.09,Z 611.91,A -85,B 0,C 180,E1 7366.882,E2 7366.882} C_VEL
LIN {X 0,Y 467.463,Z 611.91,A -85,B 0,C 180,E1 7372.553,E2 7372.553} C_VEL
LIN {X 0,Y 467.774,Z 611.91,A -85,B 0,C 180,E1 7378.142,E2 7378.142} C_VEL
LIN {X 0,Y 467.662,Z 611.91,A -85,B 0,C 180,E1 7383.709,E2 7383.709} C_VEL
LIN {X 0,Y 467.398,Z 611.91,A -85,B 0,C 180,E1 7389.317,E2 7389.317} C_VEL
LIN {X 0,Y 467.213,Z 611.91,A -85,B 0,C 180,E1 7395.021,E2 7395.021} C_VEL
LIN {X 0,Y 467.095,Z 611.91,A -85,B 0,C 180,E1 7400.884,E2 7400.884} C_VEL
LIN {X 0,Y 466.896,Z 611.91,A -85,B 0,C 180,E1 7406.995,E2 7406.995} C_VEL
LIN {X 0,Y 466.762,Z 611.91,A -85,B 0,C 180,E1 7413.46,E2 7413.46} C_VEL
LIN {X 0,Y 466.634,Z 611.91,A -85,B 0,C 180,E1 7420.454,E2 7420.454} C_VEL
LIN {X 0,Y 466.789,Z 611.91,A -85,B 0,C 180,E1 7427.067,E2 7427.067} C_VEL
LIN {X 0,Y 466.721,Z 611.91,A -85,B 0,C 180,E1 7431.949,E2 7431.949} C_VEL
LIN {X 0,Y 466.897,Z 612.422,A -85,B 0,C 180,E1 7436.154,E2 7436.154} C_VEL
LIN {X 0,Y 481.023,Z 644.057,A -85,B 0,C 180,E1 7437.823,E2 7437.823} C_VEL
LIN {X 0,Y 480.91,Z 652.495,A -85,B 0,C 180,E1 7437.989,E2 7437.989} C_VEL
LIN {X 0,Y 477.527,Z 667.33,A -85,B 0,C 180,E1 7438.158,E2 7438.158} C_VEL
LIN {X 0,Y 475.188,Z 702.567,A -85,B 0,C 180,E1 7439.493,E2 7439.493} C_VEL
LIN {X 0,Y 471.846,Z 739.55,A -85,B 0,C 180,E1 7441.701,E2 7441.701} C_VEL
LIN {X 0,Y 468.398,Z 771.944,A -85,B 0,C 180,E1 7444.514,E2 7444.514} C_VEL
LIN {X 0,Y 465.236,Z 800.424,A -85,B 0,C 180,E1 7447.868,E2 7447.868} C_VEL
LIN {X 0,Y 462.668,Z 825.416,A -85,B 0,C 180,E1 7451.88,E2 7451.88} C_VEL
LIN {X 0,Y 461.142,Z 844.259,A -85,B 0,C 180,E1 7456.053,E2 7456.053} C_VEL
LIN {X 0,Y 460.335,Z 858.495,A -85,B 0,C 180,E1 7460.612,E2 7460.612} C_VEL
LIN {X 0,Y 460.074,Z 866.909,A -85,B 0,C 180,E1 7465.281,E2 7465.281} C_VEL
LIN {X 0,Y 459.981,Z 869.835,A -85,B 0,C 180,E1 7470,E2 7470} C_VEL
LIN {X 0,Y 460.037,Z 868.025,A -85,B 0,C 180,E1 7473.774,E2 7473.774} C_VEL
LIN {X 0,Y 460.313,Z 860.545,A -85,B 0,C 180,E1 7478.472,E2 7478.472} C_VEL
LIN {X 0,Y 460.845,Z 848.46,A -85,B 0,C 180,E1 7482.813,E2 7482.813} C_VEL
LIN {X 0,Y 462.199,Z 830.351,A -85,B 0,C 180,E1 7487.147,E2 7487.147} C_VEL
LIN {X 0,Y 464.376,Z 808.221,A -85,B 0,C 180,E1 7491.017,E2 7491.017} C_VEL
LIN {X 0,Y 467.574,Z 778.896,A -85,B 0,C 180,E1 7494.767,E2 7494.767} C_VEL
LIN {X 0,Y 470.83,Z 749.397,A -85,B 0,C 180,E1 7497.534,E2 7497.534} C_VEL
LIN {X 0,Y 474.245,Z 714.054,A -85,B 0,C 180,E1 7499.923,E2 7499.923} C_VEL
LIN {X 0,Y 476.853,Z 677.095,A -85,B 0,C 180,E1 7501.545,E2 7501.545} C_VEL
LIN {X 0,Y 477.701,Z 654.933,A -85,B 0,C 180,E1 7502.191,E2 7502.191} C_VEL
LIN {X 0,Y 458.915,Z 611.91,A -85,B 0,C 180,E1 7504.627,E2 7504.627} C_VEL
LIN {X 0,Y 458.84,Z 611.91,A -85,B 0,C 180,E1 7511.296,E2 7511.296} C_VEL
LIN {X 0,Y 458.787,Z 611.91,A -85,B 0,C 180,E1 7516.554,E2 7516.554} C_VEL
LIN {X 0,Y 458.758,Z 611.91,A -85,B 0,C 180,E1 7523.56,E2 7523.56} C_VEL
LIN {X 0,Y 458.898,Z 611.91,A -85,B 0,C 180,E1 7530.342,E2 7530.342} C_VEL
LIN {X 0,Y 459.029,Z 611.91,A -85,B 0,C 180,E1 7536.688,E2 7536.688} C_VEL
LIN {X 0,Y 459.253,Z 611.91,A -85,B 0,C 180,E1 7542.953,E2 7542.953} C_VEL
LIN {X 0,Y 459.372,Z 611.91,A -85,B 0,C 180,E1 7548.598,E2 7548.598} C_VEL
LIN {X 0,Y 459.567,Z 611.91,A -85,B 0,C 180,E1 7554.332,E2 7554.332} C_VEL
LIN {X 0,Y 459.759,Z 611.91,A -85,B 0,C 180,E1 7560.003,E2 7560.003} C_VEL
LIN {X 0,Y 459.619,Z 611.91,A -85,B 0,C 180,E1 7565.675,E2 7565.675} C_VEL
LIN {X 0,Y 459.357,Z 611.91,A -85,B 0,C 180,E1 7571.409,E2 7571.409} C_VEL
LIN {X 0,Y 459.24,Z 611.91,A -85,B 0,C 180,E1 7577.263,E2 7577.263} C_VEL
LIN {X 0,Y 459.088,Z 611.91,A -85,B 0,C 180,E1 7583.316,E2 7583.316} C_VEL
LIN {X 0,Y 458.848,Z 611.91,A -85,B 0,C 180,E1 7589.669,E2 7589.669} C_VEL
LIN {X 0,Y 458.787,Z 611.91,A -85,B 0,C 180,E1 7596.446,E2 7596.446} C_VEL
LIN {X 0,Y 458.786,Z 611.91,A -85,B 0,C 180,E1 7601.304,E2 7601.304} C_VEL
LIN {X 0,Y 458.817,Z 611.91,A -85,B 0,C 180,E1 7606.553,E2 7606.553} C_VEL
LIN {X 0,Y 458.746,Z 611.91,A -85,B 0,C 180,E1 7612.385,E2 7612.385} C_VEL
LIN {X 0,Y 458.839,Z 611.91,A -85,B 0,C 180,E1 7619.088,E2 7619.088} C_VEL
LIN {X 0,Y 459.019,Z 611.91,A -85,B 0,C 180,E1 7624.609,E2 7624.609} C_VEL
LIN {X 0,Y 459.194,Z 611.91,A -85,B 0,C 180,E1 7630.748,E2 7630.748} C_VEL
LIN {X 0,Y 459.33,Z 611.91,A -85,B 0,C 180,E1 7636.66,E2 7636.66} C_VEL
LIN {X 0,Y 459.521,Z 611.91,A -85,B 0,C 180,E1 7642.427,E2 7642.427} C_VEL
LIN {X 0,Y 459.84,Z 611.91,A -85,B 0,C 180,E1 7648.113,E2 7648.113} C_VEL
LIN {X 0,Y 459.688,Z 611.91,A -85,B 0,C 180,E1 7653.777,E2 7653.777} C_VEL
LIN {X 0,Y 459.464,Z 611.91,A -85,B 0,C 180,E1 7659.483,E2 7659.483} C_VEL
LIN {X 0,Y 459.281,Z 611.91,A -85,B 0,C 180,E1 7665.291,E2 7665.291} C_VEL
LIN {X 0,Y 459.129,Z 611.91,A -85,B 0,C 180,E1 7671.269,E2 7671.269} C_VEL
LIN {X 0,Y 458.962,Z 611.91,A -85,B 0,C 180,E1 7677.506,E2 7677.506} C_VEL
LIN {X 0,Y 458.901,Z 611.91,A -85,B 0,C 180,E1 7684.117,E2 7684.117} C_VEL
LIN {X 0,Y 458.759,Z 611.91,A -85,B 0,C 180,E1 7690.615,E2 7690.615} C_VEL
LIN {X 0,Y 458.645,Z 611.91,A -85,B 0,C 180,E1 7696.573,E2 7696.573} C_VEL
LIN {X 0,Y 458.685,Z 611.91,A -85,B 0,C 180,E1 7702.392,E2 7702.392} C_VEL
LIN {X 0,Y 458.838,Z 611.91,A -85,B 0,C 180,E1 7709.086,E2 7709.086} C_VEL
LIN {X 0,Y 459.035,Z 611.91,A -85,B 0,C 180,E1 7714.607,E2 7714.607} C_VEL
LIN {X 0,Y 459.284,Z 611.91,A -85,B 0,C 180,E1 7720.749,E2 7720.749} C_VEL
LIN {X 0,Y 459.193,Z 611.91,A -85,B 0,C 180,E1 7726.653,E2 7726.653} C_VEL
LIN {X 0,Y 459.536,Z 611.91,A -85,B 0,C 180,E1 7732.424,E2 7732.424} C_VEL
LIN {X 0,Y 459.863,Z 611.91,A -85,B 0,C 180,E1 7738.11,E2 7738.11} C_VEL
LIN {X 0,Y 459.746,Z 611.91,A -85,B 0,C 180,E1 7743.773,E2 7743.773} C_VEL
LIN {X 0,Y 459.497,Z 611.91,A -85,B 0,C 180,E1 7749.479,E2 7749.479} C_VEL
LIN {X 0,Y 459.274,Z 611.91,A -85,B 0,C 180,E1 7755.287,E2 7755.287} C_VEL
LIN {X 0,Y 459.141,Z 611.91,A -85,B 0,C 180,E1 7761.264,E2 7761.264} C_VEL
LIN {X 0,Y 458.952,Z 611.91,A -85,B 0,C 180,E1 7767.502,E2 7767.502} C_VEL
LIN {X 0,Y 458.769,Z 611.91,A -85,B 0,C 180,E1 7774.122,E2 7774.122} C_VEL
LIN {X 0,Y 458.722,Z 611.91,A -85,B 0,C 180,E1 7780.612,E2 7780.612} C_VEL
LIN {X 0,Y 458.845,Z 611.91,A -85,B 0,C 180,E1 7786.539,E2 7786.539} C_VEL
LIN {X 0,Y 458.792,Z 611.91,A -85,B 0,C 180,E1 7792.366,E2 7792.366} C_VEL
LIN {X 0,Y 458.963,Z 612.184,A -85,B 0,C 180,E1 7795.488,E2 7795.488} C_VEL
LIN {X 0,Y 477.95,Z 655.468,A -85,B 0,C 180,E1 7797.839,E2 7797.839} C_VEL
LIN {X 0,Y 477.527,Z 667.33,A -85,B 0,C 180,E1 7798.158,E2 7798.158} C_VEL
LIN {X 0,Y 473.183,Z 684.19,A -85,B 0,C 180,E1 7798.442,E2 7798.442} C_VEL
LIN {X 0,Y 468.811,Z 698.545,A -85,B 0,C 180,E1 7798.818,E2 7798.818} C_VEL
LIN {X 0,Y 468.544,Z 700.571,A -85,B 0,C 180,E1 7798.912,E2 7798.912} C_VEL
LIN {X 0,Y 465.103,Z 736.167,A -85,B 0,C 180,E1 7801.013,E2 7801.013} C_VEL
LIN {X 0,Y 461.563,Z 768.106,A -85,B 0,C 180,E1 7803.715,E2 7803.715} C_VEL
LIN {X 0,Y 457.989,Z 798.181,A -85,B 0,C 180,E1 7807.205,E2 7807.205} C_VEL
LIN {X 0,Y 455.143,Z 823.385,A -85,B 0,C 180,E1 7811.232,E2 7811.232} C_VEL
LIN {X 0,Y 453.398,Z 843.039,A -85,B 0,C 180,E1 7815.537,E2 7815.537} C_VEL
LIN {X 0,Y 452.463,Z 858.052,A -85,B 0,C 180,E1 7820.368,E2 7820.368} C_VEL
LIN {X 0,Y 452.164,Z 865.507,A -85,B 0,C 180,E1 7824.235,E2 7824.235} C_VEL
LIN {X 0,Y 452.125,Z 869.151,A -85,B 0,C 180,E1 7828.081,E2 7828.081} C_VEL
LIN {X 0,Y 452.162,Z 869.152,A -85,B 0,C 180,E1 7831.919,E2 7831.919} C_VEL
LIN {X 0,Y 452.23,Z 863.928,A -85,B 0,C 180,E1 7836.729,E2 7836.729} C_VEL
LIN {X 0,Y 452.666,Z 854.25,A -85,B 0,C 180,E1 7841.088,E2 7841.088} C_VEL
LIN {X 0,Y 453.835,Z 837.895,A -85,B 0,C 180,E1 7845.727,E2 7845.727} C_VEL
LIN {X 0,Y 455.839,Z 817.098,A -85,B 0,C 180,E1 7849.904,E2 7849.904} C_VEL
LIN {X 0,Y 458.927,Z 790.178,A -85,B 0,C 180,E1 7853.831,E2 7853.831} C_VEL
LIN {X 0,Y 462.46,Z 760.392,A -85,B 0,C 180,E1 7857.017,E2 7857.017} C_VEL
LIN {X 0,Y 466.111,Z 726.413,A -85,B 0,C 180,E1 7859.659,E2 7859.659} C_VEL
LIN {X 0,Y 469.394,Z 688.988,A -85,B 0,C 180,E1 7861.594,E2 7861.594} C_VEL
LIN {X 0,Y 470.666,Z 656.476,A -85,B 0,C 180,E1 7862.686,E2 7862.686} C_VEL
LIN {X 0,Y 450.984,Z 611.91,A -85,B 0,C 180,E1 7865.243,E2 7865.243} C_VEL
LIN {X 0,Y 450.857,Z 611.91,A -85,B 0,C 180,E1 7872.193,E2 7872.193} C_VEL
LIN {X 0,Y 450.763,Z 611.91,A -85,B 0,C 180,E1 7877.803,E2 7877.803} C_VEL
LIN {X 0,Y 450.858,Z 611.91,A -85,B 0,C 180,E1 7883.703,E2 7883.703} C_VEL
LIN {X 0,Y 450.988,Z 611.91,A -85,B 0,C 180,E1 7889.768,E2 7889.768} C_VEL
LIN {X 0,Y 451.07,Z 611.91,A -85,B 0,C 180,E1 7896.252,E2 7896.252} C_VEL
LIN {X 0,Y 451.268,Z 611.91,A -85,B 0,C 180,E1 7902.429,E2 7902.429} C_VEL
LIN {X 0,Y 451.443,Z 611.91,A -85,B 0,C 180,E1 7908.395,E2 7908.395} C_VEL
LIN {X 0,Y 451.651,Z 611.91,A -85,B 0,C 180,E1 7914.232,E2 7914.232} C_VEL
LIN {X 0,Y 451.859,Z 611.91,A -85,B 0,C 180,E1 7920.003,E2 7920.003} C_VEL
LIN {X 0,Y 451.732,Z 611.91,A -85,B 0,C 180,E1 7925.774,E2 7925.774} C_VEL
LIN {X 0,Y 451.428,Z 611.91,A -85,B 0,C 180,E1 7931.612,E2 7931.612} C_VEL
LIN {X 0,Y 451.297,Z 611.91,A -85,B 0,C 180,E1 7937.577,E2 7937.577} C_VEL
LIN {X 0,Y 451.12,Z 611.91,A -85,B 0,C 180,E1 7943.753,E2 7943.753} C_VEL
LIN {X 0,Y 450.919,Z 611.91,A -85,B 0,C 180,E1 7950.245,E2 7950.245} C_VEL
LIN {X 0,Y 450.89,Z 611.91,A -85,B 0,C 180,E1 7957.19,E2 7957.19} C_VEL
LIN {X 0,Y 450.819,Z 611.91,A -85,B 0,C 180,E1 7962.366,E2 7962.366} C_VEL
LIN {X 0,Y 450.83,Z 611.91,A -85,B 0,C 180,E1 7967.804,E2 7967.804} C_VEL
LIN {X 0,Y 450.834,Z 611.91,A -85,B 0,C 180,E1 7973.71,E2 7973.71} C_VEL
LIN {X 0,Y 450.919,Z 611.91,A -85,B 0,C 180,E1 7979.758,E2 7979.758} C_VEL
LIN {X 0,Y 451.125,Z 611.91,A -85,B 0,C 180,E1 7986.25,E2 7986.25} C_VEL
LIN {X 0,Y 451.295,Z 611.91,A -85,B 0,C 180,E1 7992.426,E2 7992.426} C_VEL
LIN {X 0,Y 451.436,Z 611.91,A -85,B 0,C 180,E1 7998.391,E2 7998.391} C_VEL
LIN {X 0,Y 451.681,Z 611.91,A -85,B 0,C 180,E1 8004.228,E2 8004.228} C_VEL
LIN {X 0,Y 451.866,Z 611.91,A -85,B 0,C 180,E1 8010,E2 8010} C_VEL
LIN {X 0,Y 451.644,Z 611.91,A -85,B 0,C 180,E1 8015.772,E2 8015.772} C_VEL
LIN {X 0,Y 451.433,Z 611.91,A -85,B 0,C 180,E1 8021.609,E2 8021.609} C_VEL
LIN {X 0,Y 451.297,Z 611.91,A -85,B 0,C 180,E1 8027.574,E2 8027.574} C_VEL
LIN {X 0,Y 451.112,Z 611.91,A -85,B 0,C 180,E1 8033.75,E2 8033.75} C_VEL
LIN {X 0,Y 450.994,Z 611.91,A -85,B 0,C 180,E1 8040.237,E2 8040.237} C_VEL
LIN {X 0,Y 450.944,Z 611.91,A -85,B 0,C 180,E1 8047.182,E2 8047.182} C_VEL
LIN {X 0,Y 450.719,Z 611.91,A -85,B 0,C 180,E1 8052.349,E2 8052.349} C_VEL
LIN {X 0,Y 450.665,Z 611.91,A -85,B 0,C 180,E1 8057.782,E2 8057.782} C_VEL
LIN {X 0,Y 450.787,Z 611.91,A -85,B 0,C 180,E1 8063.715,E2 8063.715} C_VEL
LIN {X 0,Y 450.918,Z 611.91,A -85,B 0,C 180,E1 8069.755,E2 8069.755} C_VEL
LIN {X 0,Y 451.151,Z 611.91,A -85,B 0,C 180,E1 8076.249,E2 8076.249} C_VEL
LIN {X 0,Y 451.341,Z 611.91,A -85,B 0,C 180,E1 8082.425,E2 8082.425} C_VEL
LIN {X 0,Y 451.338,Z 611.91,A -85,B 0,C 180,E1 8088.385,E2 8088.385} C_VEL
LIN {X 0,Y 451.734,Z 611.91,A -85,B 0,C 180,E1 8094.226,E2 8094.226} C_VEL
LIN {X 0,Y 451.946,Z 611.91,A -85,B 0,C 180,E1 8099.997,E2 8099.997} C_VEL
LIN {X 0,Y 451.652,Z 611.91,A -85,B 0,C 180,E1 8105.768,E2 8105.768} C_VEL
LIN {X 0,Y 451.444,Z 611.91,A -85,B 0,C 180,E1 8111.605,E2 8111.605} C_VEL
LIN {X 0,Y 451.29,Z 611.91,A -85,B 0,C 180,E1 8117.57,E2 8117.57} C_VEL
LIN {X 0,Y 451.126,Z 611.91,A -85,B 0,C 180,E1 8123.745,E2 8123.745} C_VEL
LIN {X 0,Y 450.915,Z 611.91,A -85,B 0,C 180,E1 8130.237,E2 8130.237} C_VEL
LIN {X 0,Y 450.82,Z 611.91,A -85,B 0,C 180,E1 8137.188,E2 8137.188} C_VEL
LIN {X 0,Y 450.771,Z 611.91,A -85,B 0,C 180,E1 8142.359,E2 8142.359} C_VEL
LIN {X 0,Y 450.874,Z 611.91,A -85,B 0,C 180,E1 8147.809,E2 8147.809} C_VEL
LIN {X 0,Y 451.006,Z 611.91,A -85,B 0,C 180,E1 8154.759,E2 8154.759} C_VEL
LIN {X 0,Y 471.2,Z 657.817,A -85,B 0,C 180,E1 8157.396,E2 8157.396} C_VEL
LIN {X 0,Y 468.773,Z 697.115,A -85,B 0,C 180,E1 8158.751,E2 8158.751} C_VEL
LIN {X 0,Y 468.544,Z 700.571,A -85,B 0,C 180,E1 8158.912,E2 8158.912} C_VEL
LIN {X 0,Y 463.638,Z 716.824,A -85,B 0,C 180,E1 8159.53,E2 8159.53} C_VEL
LIN {X 0,Y 458.519,Z 732.27,A -85,B 0,C 180,E1 8160.271,E2 8160.271} C_VEL
LIN {X 0,Y 454.652,Z 765.473,A -85,B 0,C 180,E1 8163.017,E2 8163.017} C_VEL
LIN {X 0,Y 450.733,Z 796.202,A -85,B 0,C 180,E1 8166.577,E2 8166.577} C_VEL
LIN {X 0,Y 447.897,Z 819.647,A -85,B 0,C 180,E1 8170.243,E2 8170.243} C_VEL
LIN {X 0,Y 445.731,Z 840.827,A -85,B 0,C 180,E1 8174.758,E2 8174.758} C_VEL
LIN {X 0,Y 444.709,Z 855.282,A -85,B 0,C 180,E1 8179.208,E2 8179.208} C_VEL
LIN {X 0,Y 444.376,Z 863.694,A -85,B 0,C 180,E1 8183.151,E2 8183.151} C_VEL
LIN {X 0,Y 444.223,Z 868.918,A -85,B 0,C 180,E1 8188.047,E2 8188.047} C_VEL
LIN {X 0,Y 444.26,Z 868.919,A -85,B 0,C 180,E1 8191.953,E2 8191.953} C_VEL
LIN {X 0,Y 444.352,Z 863.693,A -85,B 0,C 180,E1 8196.849,E2 8196.849} C_VEL
LIN {X 0,Y 444.814,Z 854.014,A -85,B 0,C 180,E1 8201.287,E2 8201.287} C_VEL
LIN {X 0,Y 446.047,Z 837.656,A -85,B 0,C 180,E1 8206.009,E2 8206.009} C_VEL
LIN {X 0,Y 448.208,Z 816.858,A -85,B 0,C 180,E1 8210.258,E2 8210.258} C_VEL
LIN {X 0,Y 451.723,Z 788.737,A -85,B 0,C 180,E1 8214.402,E2 8214.402} C_VEL
LIN {X 0,Y 455.414,Z 758.803,A -85,B 0,C 180,E1 8217.604,E2 8217.604} C_VEL
LIN {X 0,Y 459.12,Z 726.409,A -85,B 0,C 180,E1 8220.141,E2 8220.141} C_VEL
LIN {X 0,Y 462.617,Z 688.752,A -85,B 0,C 180,E1 8222.111,E2 8222.111} C_VEL
LIN {X 0,Y 464.057,Z 659.25,A -85,B 0,C 180,E1 8223.117,E2 8223.117} C_VEL
LIN {X 0,Y 444.89,Z 616.948,A -85,B 0,C 180,E1 8225.665,E2 8225.665} C_VEL
LIN {X 0,Y 443.009,Z 611.91,A -85,B 0,C 180,E1 8226.036,E2 8226.036} C_VEL
LIN {X 0,Y 442.857,Z 611.91,A -85,B 0,C 180,E1 8233.139,E2 8233.139} C_VEL
LIN {X 0,Y 442.8,Z 611.91,A -85,B 0,C 180,E1 8239.491,E2 8239.491} C_VEL
LIN {X 0,Y 442.965,Z 611.91,A -85,B 0,C 180,E1 8245.117,E2 8245.117} C_VEL
LIN {X 0,Y 443.054,Z 611.91,A -85,B 0,C 180,E1 8251.423,E2 8251.423} C_VEL
LIN {X 0,Y 443.176,Z 611.91,A -85,B 0,C 180,E1 8257.931,E2 8257.931} C_VEL
LIN {X 0,Y 443.393,Z 611.91,A -85,B 0,C 180,E1 8264.151,E2 8264.151} C_VEL
LIN {X 0,Y 443.651,Z 611.91,A -85,B 0,C 180,E1 8270.179,E2 8270.179} C_VEL
LIN {X 0,Y 443.857,Z 611.91,A -85,B 0,C 180,E1 8276.092,E2 8276.092} C_VEL
LIN {X 0,Y 444.053,Z 611.91,A -85,B 0,C 180,E1 8281.957,E2 8281.957} C_VEL
LIN {X 0,Y 443.67,Z 611.91,A -85,B 0,C 180,E1 8288.252,E2 8288.252} C_VEL
LIN {X 0,Y 443.472,Z 611.91,A -85,B 0,C 180,E1 8293.83,E2 8293.83} C_VEL
LIN {X 0,Y 443.325,Z 611.91,A -85,B 0,C 180,E1 8299.973,E2 8299.973} C_VEL
LIN {X 0,Y 443.103,Z 611.91,A -85,B 0,C 180,E1 8306.375,E2 8306.375} C_VEL
LIN {X 0,Y 442.927,Z 611.91,A -85,B 0,C 180,E1 8313.159,E2 8313.159} C_VEL
LIN {X 0,Y 442.901,Z 611.91,A -85,B 0,C 180,E1 8318.163,E2 8318.163} C_VEL
LIN {X 0,Y 442.838,Z 611.91,A -85,B 0,C 180,E1 8324.112,E2 8324.112} C_VEL
LIN {X 0,Y 442.856,Z 611.91,A -85,B 0,C 180,E1 8329.49,E2 8329.49} C_VEL
LIN {X 0,Y 442.916,Z 611.91,A -85,B 0,C 180,E1 8335.129,E2 8335.129} C_VEL
LIN {X 0,Y 443.031,Z 611.91,A -85,B 0,C 180,E1 8341.416,E2 8341.416} C_VEL
LIN {X 0,Y 443.235,Z 611.91,A -85,B 0,C 180,E1 8347.929,E2 8347.929} C_VEL
LIN {X 0,Y 443.394,Z 611.91,A -85,B 0,C 180,E1 8354.147,E2 8354.147} C_VEL
LIN {X 0,Y 443.594,Z 611.91,A -85,B 0,C 180,E1 8360.174,E2 8360.174} C_VEL
LIN {X 0,Y 443.769,Z 611.91,A -85,B 0,C 180,E1 8366.087,E2 8366.087} C_VEL
LIN {X 0,Y 443.889,Z 611.91,A -85,B 0,C 180,E1 8371.955,E2 8371.955} C_VEL
LIN {X 0,Y 443.632,Z 611.91,A -85,B 0,C 180,E1 8378.21,E2 8378.21} C_VEL
LIN {X 0,Y 443.481,Z 611.91,A -85,B 0,C 180,E1 8383.826,E2 8383.826} C_VEL
LIN {X 0,Y 443.331,Z 611.91,A -85,B 0,C 180,E1 8389.969,E2 8389.969} C_VEL
LIN {X 0,Y 443.111,Z 611.91,A -85,B 0,C 180,E1 8396.372,E2 8396.372} C_VEL
LIN {X 0,Y 443.046,Z 611.91,A -85,B 0,C 180,E1 8403.146,E2 8403.146} C_VEL
LIN {X 0,Y 442.935,Z 611.91,A -85,B 0,C 180,E1 8408.166,E2 8408.166} C_VEL
LIN {X 0,Y 442.708,Z 611.91,A -85,B 0,C 180,E1 8414.092,E2 8414.092} C_VEL
LIN {X 0,Y 442.725,Z 611.91,A -85,B 0,C 180,E1 8419.473,E2 8419.473} C_VEL
LIN {X 0,Y 442.889,Z 611.91,A -85,B 0,C 180,E1 8425.131,E2 8425.131} C_VEL
LIN {X 0,Y 443.029,Z 611.91,A -85,B 0,C 180,E1 8431.413,E2 8431.413} C_VEL
LIN {X 0,Y 443.292,Z 611.91,A -85,B 0,C 180,E1 8437.929,E2 8437.929} C_VEL
LIN {X 0,Y 443.338,Z 611.91,A -85,B 0,C 180,E1 8444.142,E2 8444.142} C_VEL
LIN {X 0,Y 443.53,Z 611.91,A -85,B 0,C 180,E1 8450.169,E2 8450.169} C_VEL
LIN {X 0,Y 443.806,Z 611.91,A -85,B 0,C 180,E1 8456.084,E2 8456.084} C_VEL
LIN {X 0,Y 443.889,Z 611.91,A -85,B 0,C 180,E1 8461.951,E2 8461.951} C_VEL
LIN {X 0,Y 443.64,Z 611.91,A -85,B 0,C 180,E1 8468.226,E2 8468.226} C_VEL
LIN {X 0,Y 443.471,Z 611.91,A -85,B 0,C 180,E1 8473.823,E2 8473.823} C_VEL
LIN {X 0,Y 443.336,Z 611.91,A -85,B 0,C 180,E1 8479.965,E2 8479.965} C_VEL
LIN {X 0,Y 443.108,Z 611.91,A -85,B 0,C 180,E1 8486.367,E2 8486.367} C_VEL
LIN {X 0,Y 442.93,Z 611.91,A -85,B 0,C 180,E1 8493.15,E2 8493.15} C_VEL
LIN {X 0,Y 442.838,Z 611.91,A -85,B 0,C 180,E1 8498.153,E2 8498.153} C_VEL
LIN {X 0,Y 442.85,Z 611.91,A -85,B 0,C 180,E1 8504.113,E2 8504.113} C_VEL
LIN {X 0,Y 442.888,Z 611.91,A -85,B 0,C 180,E1 8509.494,E2 8509.494} C_VEL
LIN {X 0,Y 443.035,Z 611.91,A -85,B 0,C 180,E1 8514.032,E2 8514.032} C_VEL
LIN {X 0,Y 464.473,Z 660.265,A -85,B 0,C 180,E1 8516.947,E2 8516.947} C_VEL
LIN {X 0,Y 461.879,Z 698.445,A -85,B 0,C 180,E1 8518.307,E2 8518.307} C_VEL
LIN {X 0,Y 458.519,Z 732.27,A -85,B 0,C 180,E1 8520.271,E2 8520.271} C_VEL
LIN {X 0,Y 453.189,Z 747.5,A -85,B 0,C 180,E1 8521.181,E2 8521.181} C_VEL
LIN {X 0,Y 447.882,Z 761.849,A -85,B 0,C 180,E1 8522.224,E2 8522.224} C_VEL
LIN {X 0,Y 444.038,Z 790.496,A -85,B 0,C 180,E1 8525.431,E2 8525.431} C_VEL
LIN {X 0,Y 440.617,Z 816.619,A -85,B 0,C 180,E1 8529.377,E2 8529.377} C_VEL
LIN {X 0,Y 438.291,Z 837.417,A -85,B 0,C 180,E1 8533.7,E2 8533.7} C_VEL
LIN {X 0,Y 436.995,Z 852.325,A -85,B 0,C 180,E1 8538.002,E2 8538.002} C_VEL
LIN {X 0,Y 436.573,Z 861.803,A -85,B 0,C 180,E1 8542.026,E2 8542.026} C_VEL
LIN {X 0,Y 436.336,Z 867.323,A -85,B 0,C 180,E1 8546.021,E2 8546.021} C_VEL
LIN {X 0,Y 436.308,Z 869.136,A -85,B 0,C 180,E1 8550,E2 8550} C_VEL
LIN {X 0,Y 436.36,Z 867.324,A -85,B 0,C 180,E1 8553.979,E2 8553.979} C_VEL
LIN {X 0,Y 436.626,Z 860.553,A -85,B 0,C 180,E1 8558.585,E2 8558.585} C_VEL
LIN {X 0,Y 437.378,Z 847.747,A -85,B 0,C 180,E1 8563.513,E2 8563.513} C_VEL
LIN {X 0,Y 439.081,Z 829.634,A -85,B 0,C 180,E1 8568.08,E2 8568.08} C_VEL
LIN {X 0,Y 441.767,Z 807.502,A -85,B 0,C 180,E1 8572.148,E2 8572.148} C_VEL
LIN {X 0,Y 445.686,Z 778.227,A -85,B 0,C 180,E1 8576.066,E2 8576.066} C_VEL
LIN {X 0,Y 449.764,Z 747.586,A -85,B 0,C 180,E1 8579.041,E2 8579.041} C_VEL
LIN {X 0,Y 453.722,Z 712.891,A -85,B 0,C 180,E1 8581.457,E2 8581.457} C_VEL
LIN {X 0,Y 456.858,Z 675.041,A -85,B 0,C 180,E1 8583.153,E2 8583.153} C_VEL
LIN {X 0,Y 457.193,Z 661.397,A -85,B 0,C 180,E1 8583.604,E2 8583.604} C_VEL
LIN {X 0,Y 440.097,Z 623.263,A -85,B 0,C 180,E1 8585.986,E2 8585.986} C_VEL
LIN {X 0,Y 435.111,Z 611.91,A -85,B 0,C 180,E1 8586.771,E2 8586.771} C_VEL
LIN {X 0,Y 434.972,Z 611.91,A -85,B 0,C 180,E1 8594.12,E2 8594.12} C_VEL
LIN {X 0,Y 434.871,Z 611.91,A -85,B 0,C 180,E1 8601.2,E2 8601.2} C_VEL
LIN {X 0,Y 435.08,Z 611.91,A -85,B 0,C 180,E1 8606.635,E2 8606.635} C_VEL
LIN {X 0,Y 435.167,Z 611.91,A -85,B 0,C 180,E1 8613.114,E2 8613.114} C_VEL
LIN {X 0,Y 435.36,Z 611.91,A -85,B 0,C 180,E1 8619.881,E2 8619.881} C_VEL
LIN {X 0,Y 435.543,Z 611.91,A -85,B 0,C 180,E1 8626.742,E2 8626.742} C_VEL
LIN {X 0,Y 435.783,Z 611.91,A -85,B 0,C 180,E1 8632.016,E2 8632.016} C_VEL
LIN {X 0,Y 435.996,Z 611.91,A -85,B 0,C 180,E1 8638.014,E2 8638.014} C_VEL
LIN {X 0,Y 435.896,Z 611.91,A -85,B 0,C 180,E1 8643.987,E2 8643.987} C_VEL
LIN {X 0,Y 435.66,Z 611.91,A -85,B 0,C 180,E1 8650.01,E2 8650.01} C_VEL
LIN {X 0,Y 435.501,Z 611.91,A -85,B 0,C 180,E1 8656.152,E2 8656.152} C_VEL
LIN {X 0,Y 435.305,Z 611.91,A -85,B 0,C 180,E1 8662.498,E2 8662.498} C_VEL
LIN {X 0,Y 435.03,Z 611.91,A -85,B 0,C 180,E1 8669.163,E2 8669.163} C_VEL
LIN {X 0,Y 435.012,Z 611.91,A -85,B 0,C 180,E1 8673.843,E2 8673.843} C_VEL
LIN {X 0,Y 434.926,Z 611.91,A -85,B 0,C 180,E1 8680.017,E2 8680.017} C_VEL
LIN {X 0,Y 434.928,Z 611.91,A -85,B 0,C 180,E1 8686.977,E2 8686.977} C_VEL
LIN {X 0,Y 434.896,Z 611.91,A -85,B 0,C 180,E1 8693.712,E2 8693.712} C_VEL
LIN {X 0,Y 435.007,Z 611.91,A -85,B 0,C 180,E1 8698.528,E2 8698.528} C_VEL
LIN {X 0,Y 435.226,Z 611.91,A -85,B 0,C 180,E1 8705.326,E2 8705.326} C_VEL
LIN {X 0,Y 435.423,Z 611.91,A -85,B 0,C 180,E1 8711.763,E2 8711.763} C_VEL
LIN {X 0,Y 435.585,Z 611.91,A -85,B 0,C 180,E1 8717.962,E2 8717.962} C_VEL
LIN {X 0,Y 435.847,Z 611.91,A -85,B 0,C 180,E1 8724.018,E2 8724.018} C_VEL
LIN {X 0,Y 436.079,Z 611.91,A -85,B 0,C 180,E1 8730,E2 8730} C_VEL
LIN {X 0,Y 435.811,Z 611.91,A -85,B 0,C 180,E1 8735.982,E2 8735.982} C_VEL
LIN {X 0,Y 435.583,Z 611.91,A -85,B 0,C 180,E1 8742.038,E2 8742.038} C_VEL
LIN {X 0,Y 435.429,Z 611.91,A -85,B 0,C 180,E1 8748.237,E2 8748.237} C_VEL
LIN {X 0,Y 435.175,Z 611.91,A -85,B 0,C 180,E1 8755.229,E2 8755.229} C_VEL
LIN {X 0,Y 435.114,Z 611.91,A -85,B 0,C 180,E1 8761.463,E2 8761.463} C_VEL
LIN {X 0,Y 435.001,Z 611.91,A -85,B 0,C 180,E1 8766.816,E2 8766.816} C_VEL
LIN {X 0,Y 434.807,Z 611.91,A -85,B 0,C 180,E1 8773.006,E2 8773.006} C_VEL
LIN {X 0,Y 434.797,Z 611.91,A -85,B 0,C 180,E1 8780.004,E2 8780.004} C_VEL
LIN {X 0,Y 434.999,Z 611.91,A -85,B 0,C 180,E1 8786.651,E2 8786.651} C_VEL
LIN {X 0,Y 435.18,Z 611.91,A -85,B 0,C 180,E1 8793.107,E2 8793.107} C_VEL
LIN {X 0,Y 435.465,Z 611.91,A -85,B 0,C 180,E1 8799.843,E2 8799.843} C_VEL
LIN {X 0,Y 435.419,Z 611.91,A -85,B 0,C 180,E1 8806.812,E2 8806.812} C_VEL
LIN {X 0,Y 435.794,Z 611.91,A -85,B 0,C 180,E1 8812.008,E2 8812.008} C_VEL
LIN {X 0,Y 436.171,Z 611.91,A -85,B 0,C 180,E1 8818.007,E2 8818.007} C_VEL
LIN {X 0,Y 436.014,Z 611.91,A -85,B 0,C 180,E1 8823.979,E2 8823.979} C_VEL
LIN {X 0,Y 435.715,Z 611.91,A -85,B 0,C 180,E1 8830.001,E2 8830.001} C_VEL
LIN {X 0,Y 435.503,Z 611.91,A -85,B 0,C 180,E1 8836.144,E2 8836.144} C_VEL
LIN {X 0,Y 435.312,Z 611.91,A -85,B 0,C 180,E1 8842.489,E2 8842.489} C_VEL
LIN {X 0,Y 435.03,Z 611.91,A -85,B 0,C 180,E1 8849.154,E2 8849.154} C_VEL
LIN {X 0,Y 434.999,Z 611.91,A -85,B 0,C 180,E1 8853.835,E2 8853.835} C_VEL
LIN {X 0,Y 434.863,Z 611.91,A -85,B 0,C 180,E1 8860.007,E2 8860.007} C_VEL
LIN {X 0,Y 434.985,Z 611.91,A -85,B 0,C 180,E1 8865.882,E2 8865.882} C_VEL
LIN {X 0,Y 435.127,Z 611.91,A -85,B 0,C 180,E1 8873.298,E2 8873.298} C_VEL
LIN {X 0,Y 443.589,Z 630.188,A -85,B 0,C 180,E1 8874.473,E2 8874.473} C_VEL
LIN {X 0,Y 457.689,Z 663.097,A -85,B 0,C 180,E1 8876.49,E2 8876.49} C_VEL
LIN {X 0,Y 455.017,Z 699.31,A -85,B 0,C 180,E1 8877.833,E2 8877.833} C_VEL
LIN {X 0,Y 451.175,Z 735.297,A -85,B 0,C 180,E1 8879.997,E2 8879.997} C_VEL
LIN {X 0,Y 447.882,Z 761.849,A -85,B 0,C 180,E1 8882.224,E2 8882.224} C_VEL
LIN {X 0,Y 442.388,Z 775.766,A -85,B 0,C 180,E1 8883.412,E2 8883.412} C_VEL
LIN {X 0,Y 437.217,Z 787.148,A -85,B 0,C 180,E1 8884.575,E2 8884.575} C_VEL
LIN {X 0,Y 436.915,Z 788.684,A -85,B 0,C 180,E1 8884.776,E2 8884.776} C_VEL
LIN {X 0,Y 433.077,Z 816.38,A -85,B 0,C 180,E1 8889.001,E2 8889.001} C_VEL
LIN {X 0,Y 430.535,Z 837.178,A -85,B 0,C 180,E1 8893.397,E2 8893.397} C_VEL
LIN {X 0,Y 429.151,Z 852.088,A -85,B 0,C 180,E1 8897.779,E2 8897.779} C_VEL
LIN {X 0,Y 428.679,Z 861.568,A -85,B 0,C 180,E1 8901.878,E2 8901.878} C_VEL
LIN {X 0,Y 428.438,Z 867.089,A -85,B 0,C 180,E1 8905.947,E2 8905.947} C_VEL
LIN {X 0,Y 428.412,Z 868.902,A -85,B 0,C 180,E1 8910,E2 8910} C_VEL
LIN {X 0,Y 428.463,Z 867.09,A -85,B 0,C 180,E1 8914.053,E2 8914.053} C_VEL
LIN {X 0,Y 428.747,Z 860.542,A -85,B 0,C 180,E1 8918.632,E2 8918.632} C_VEL
LIN {X 0,Y 429.419,Z 849.051,A -85,B 0,C 180,E1 8923.249,E2 8923.249} C_VEL
LIN {X 0,Y 431.102,Z 831.746,A -85,B 0,C 180,E1 8927.897,E2 8927.897} C_VEL
LIN {X 0,Y 434.048,Z 808.859,A -85,B 0,C 180,E1 8932.293,E2 8932.293} C_VEL
LIN {X 0,Y 438.037,Z 780.728,A -85,B 0,C 180,E1 8936.201,E2 8936.201} C_VEL
LIN {X 0,Y 442.322,Z 750.715,A -85,B 0,C 180,E1 8939.268,E2 8939.268} C_VEL
LIN {X 0,Y 446.586,Z 715.133,A -85,B 0,C 180,E1 8941.844,E2 8941.844} C_VEL
LIN {X 0,Y 449.933,Z 678.346,A -85,B 0,C 180,E1 8943.583,E2 8943.583} C_VEL
LIN {X 0,Y 450.596,Z 663.904,A -85,B 0,C 180,E1 8944.075,E2 8944.075} C_VEL
LIN {X 0,Y 433.516,Z 625.767,A -85,B 0,C 180,E1 8946.565,E2 8946.565} C_VEL
LIN {X 0,Y 427.159,Z 612.963,A -85,B 0,C 180,E1 8947.46,E2 8947.46} C_VEL
LIN {X 0,Y 427.093,Z 611.91,A -85,B 0,C 180,E1 8947.619,E2 8947.619} C_VEL
LIN {X 0,Y 427.031,Z 611.91,A -85,B 0,C 180,E1 8952.35,E2 8952.35} C_VEL
LIN {X 0,Y 426.954,Z 611.91,A -85,B 0,C 180,E1 8958.133,E2 8958.133} C_VEL
LIN {X 0,Y 426.978,Z 611.91,A -85,B 0,C 180,E1 8964.644,E2 8964.644} C_VEL
LIN {X 0,Y 427.172,Z 611.91,A -85,B 0,C 180,E1 8970.256,E2 8970.256} C_VEL
LIN {X 0,Y 427.308,Z 611.91,A -85,B 0,C 180,E1 8977.108,E2 8977.108} C_VEL
LIN {X 0,Y 427.54,Z 611.91,A -85,B 0,C 180,E1 8983.547,E2 8983.547} C_VEL
LIN {X 0,Y 427.78,Z 611.91,A -85,B 0,C 180,E1 8989.811,E2 8989.811} C_VEL
LIN {X 0,Y 428.027,Z 611.91,A -85,B 0,C 180,E1 8995.947,E2 8995.947} C_VEL
LIN {X 0,Y 428.256,Z 611.91,A -85,B 0,C 180,E1 9002.03,E2 9002.03} C_VEL
LIN {X 0,Y 427.891,Z 611.91,A -85,B 0,C 180,E1 9008.14,E2 9008.14} C_VEL
LIN {X 0,Y 427.603,Z 611.91,A -85,B 0,C 180,E1 9014.354,E2 9014.354} C_VEL
LIN {X 0,Y 427.408,Z 611.91,A -85,B 0,C 180,E1 9020.75,E2 9020.75} C_VEL
LIN {X 0,Y 427.152,Z 611.91,A -85,B 0,C 180,E1 9027.609,E2 9027.609} C_VEL
LIN {X 0,Y 427.078,Z 611.91,A -85,B 0,C 180,E1 9032.128,E2 9032.128} C_VEL
LIN {X 0,Y 427.027,Z 611.91,A -85,B 0,C 180,E1 9038.737,E2 9038.737} C_VEL
LIN {X 0,Y 427.013,Z 611.91,A -85,B 0,C 180,E1 9045.168,E2 9045.168} C_VEL
LIN {X 0,Y 426.991,Z 611.91,A -85,B 0,C 180,E1 9051.272,E2 9051.272} C_VEL
LIN {X 0,Y 427.11,Z 611.91,A -85,B 0,C 180,E1 9058.299,E2 9058.299} C_VEL
LIN {X 0,Y 427.304,Z 611.91,A -85,B 0,C 180,E1 9064.837,E2 9064.837} C_VEL
LIN {X 0,Y 427.485,Z 611.91,A -85,B 0,C 180,E1 9071.412,E2 9071.412} C_VEL
LIN {X 0,Y 427.664,Z 611.91,A -85,B 0,C 180,E1 9077.736,E2 9077.736} C_VEL
LIN {X 0,Y 427.93,Z 611.91,A -85,B 0,C 180,E1 9083.907,E2 9083.907} C_VEL
LIN {X 0,Y 428.178,Z 611.91,A -85,B 0,C 180,E1 9090,E2 9090} C_VEL
LIN {X 0,Y 427.895,Z 611.91,A -85,B 0,C 180,E1 9096.093,E2 9096.093} C_VEL
LIN {X 0,Y 427.663,Z 611.91,A -85,B 0,C 180,E1 9102.264,E2 9102.264} C_VEL
LIN {X 0,Y 427.488,Z 611.91,A -85,B 0,C 180,E1 9108.588,E2 9108.588} C_VEL
LIN {X 0,Y 427.292,Z 611.91,A -85,B 0,C 180,E1 9115.164,E2 9115.164} C_VEL
LIN {X 0,Y 427.181,Z 611.91,A -85,B 0,C 180,E1 9122.117,E2 9122.117} C_VEL
LIN {X 0,Y 427.043,Z 611.91,A -85,B 0,C 180,E1 9128.737,E2 9128.737} C_VEL
LIN {X 0,Y 426.847,Z 611.91,A -85,B 0,C 180,E1 9135.187,E2 9135.187} C_VEL
LIN {X 0,Y 426.89,Z 611.91,A -85,B 0,C 180,E1 9141.286,E2 9141.286} C_VEL
LIN {X 0,Y 427.105,Z 611.91,A -85,B 0,C 180,E1 9148.297,E2 9148.297} C_VEL
LIN {X 0,Y 427.319,Z 611.91,A -85,B 0,C 180,E1 9154.835,E2 9154.835} C_VEL
LIN {X 0,Y 427.557,Z 611.91,A -85,B 0,C 180,E1 9161.412,E2 9161.412} C_VEL
LIN {X 0,Y 427.561,Z 611.91,A -85,B 0,C 180,E1 9167.73,E2 9167.73} C_VEL
LIN {X 0,Y 427.974,Z 611.91,A -85,B 0,C 180,E1 9173.904,E2 9173.904} C_VEL
LIN {X 0,Y 428.248,Z 611.91,A -85,B 0,C 180,E1 9179.996,E2 9179.996} C_VEL
LIN {X 0,Y 427.902,Z 611.91,A -85,B 0,C 180,E1 9186.089,E2 9186.089} C_VEL
LIN {X 0,Y 427.666,Z 611.91,A -85,B 0,C 180,E1 9192.26,E2 9192.26} C_VEL
LIN {X 0,Y 427.486,Z 611.91,A -85,B 0,C 180,E1 9198.583,E2 9198.583} C_VEL
LIN {X 0,Y 427.295,Z 611.91,A -85,B 0,C 180,E1 9205.158,E2 9205.158} C_VEL
LIN {X 0,Y 427.074,Z 611.91,A -85,B 0,C 180,E1 9212.12,E2 9212.12} C_VEL
LIN {X 0,Y 426.966,Z 611.91,A -85,B 0,C 180,E1 9218.727,E2 9218.727} C_VEL
LIN {X 0,Y 427.032,Z 611.91,A -85,B 0,C 180,E1 9225.155,E2 9225.155} C_VEL
LIN {X 0,Y 427.076,Z 611.91,A -85,B 0,C 180,E1 9232.227,E2 9232.227} C_VEL
LIN {X 0,Y 427.125,Z 611.91,A -85,B 0,C 180,E1 9232.504,E2 9232.504} C_VEL
LIN {X 0,Y 433.818,Z 626.281,A -85,B 0,C 180,E1 9233.474,E2 9233.474} C_VEL
LIN {X 0,Y 450.842,Z 664.567,A -85,B 0,C 180,E1 9235.968,E2 9235.968} C_VEL
LIN {X 0,Y 448.103,Z 700.888,A -85,B 0,C 180,E1 9237.385,E2 9237.385} C_VEL
LIN {X 0,Y 444.013,Z 737.058,A -85,B 0,C 180,E1 9239.624,E2 9239.624} C_VEL
LIN {X 0,Y 439.821,Z 768.587,A -85,B 0,C 180,E1 9242.447,E2 9242.447} C_VEL
LIN {X 0,Y 436.915,Z 788.684,A -85,B 0,C 180,E1 9244.776,E2 9244.776} C_VEL
LIN {X 0,Y 431.492,Z 800.915,A -85,B 0,C 180,E1 9246.288,E2 9246.288} C_VEL
LIN {X 0,Y 426.047,Z 812.182,A -85,B 0,C 180,E1 9247.917,E2 9247.917} C_VEL
LIN {X 0,Y 423.19,Z 833.841,A -85,B 0,C 180,E1 9252.296,E2 9252.296} C_VEL
LIN {X 0,Y 421.433,Z 850.499,A -85,B 0,C 180,E1 9257.082,E2 9257.082} C_VEL
LIN {X 0,Y 420.801,Z 861.333,A -85,B 0,C 180,E1 9261.725,E2 9261.725} C_VEL
LIN {X 0,Y 420.551,Z 866.856,A -85,B 0,C 180,E1 9265.871,E2 9265.871} C_VEL
LIN {X 0,Y 420.532,Z 868.669,A -85,B 0,C 180,E1 9270,E2 9270} C_VEL
LIN {X 0,Y 420.574,Z 866.856,A -85,B 0,C 180,E1 9274.129,E2 9274.129} C_VEL
LIN {X 0,Y 420.849,Z 860.306,A -85,B 0,C 180,E1 9278.795,E2 9278.795} C_VEL
LIN {X 0,Y 421.696,Z 847.806,A -85,B 0,C 180,E1 9283.847,E2 9283.847} C_VEL
LIN {X 0,Y 423.704,Z 829.156,A -85,B 0,C 180,E1 9288.76,E2 9288.76} C_VEL
LIN {X 0,Y 426.821,Z 807.024,A -85,B 0,C 180,E1 9292.967,E2 9292.967} C_VEL
LIN {X 0,Y 431.076,Z 778.561,A -85,B 0,C 180,E1 9296.912,E2 9296.912} C_VEL
LIN {X 0,Y 435.659,Z 747.755,A -85,B 0,C 180,E1 9300.016,E2 9300.016} C_VEL
LIN {X 0,Y 440.135,Z 712.883,A -85,B 0,C 180,E1 9302.513,E2 9302.513} C_VEL
LIN {X 0,Y 443.55,Z 675.793,A -85,B 0,C 180,E1 9304.231,E2 9304.231} C_VEL
LIN {X 0,Y 443.728,Z 665.784,A -85,B 0,C 180,E1 9304.606,E2 9304.606} C_VEL
LIN {X 0,Y 427.192,Z 628.723,A -85,B 0,C 180,E1 9307.131,E2 9307.131} C_VEL
LIN {X 0,Y 419.298,Z 613.456,A -85,B 0,C 180,E1 9308.271,E2 9308.271} C_VEL
LIN {X 0,Y 419.149,Z 611.91,A -85,B 0,C 180,E1 9308.341,E2 9308.341} C_VEL
LIN {X 0,Y 419.028,Z 611.91,A -85,B 0,C 180,E1 9313.734,E2 9313.734} C_VEL
LIN {X 0,Y 418.994,Z 611.91,A -85,B 0,C 180,E1 9319.432,E2 9319.432} C_VEL
LIN {X 0,Y 419.094,Z 611.91,A -85,B 0,C 180,E1 9326.193,E2 9326.193} C_VEL
LIN {X 0,Y 419.255,Z 611.91,A -85,B 0,C 180,E1 9332.006,E2 9332.006} C_VEL
LIN {X 0,Y 419.439,Z 611.91,A -85,B 0,C 180,E1 9338.845,E2 9338.845} C_VEL
LIN {X 0,Y 419.685,Z 611.91,A -85,B 0,C 180,E1 9345.377,E2 9345.377} C_VEL
LIN {X 0,Y 419.951,Z 611.91,A -85,B 0,C 180,E1 9351.712,E2 9351.712} C_VEL
LIN {X 0,Y 420.182,Z 611.91,A -85,B 0,C 180,E1 9357.939,E2 9357.939} C_VEL
LIN {X 0,Y 420.083,Z 611.91,A -85,B 0,C 180,E1 9364.137,E2 9364.137} C_VEL
LIN {X 0,Y 419.803,Z 611.91,A -85,B 0,C 180,E1 9370.392,E2 9370.392} C_VEL
LIN {X 0,Y 419.635,Z 611.91,A -85,B 0,C 180,E1 9376.78,E2 9376.78} C_VEL
LIN {X 0,Y 419.388,Z 611.91,A -85,B 0,C 180,E1 9383.401,E2 9383.401} C_VEL
LIN {X 0,Y 419.187,Z 611.91,A -85,B 0,C 180,E1 9390.378,E2 9390.378} C_VEL
LIN {X 0,Y 419.092,Z 611.91,A -85,B 0,C 180,E1 9397.364,E2 9397.364} C_VEL
LIN {X 0,Y 419.005,Z 611.91,A -85,B 0,C 180,E1 9403.723,E2 9403.723} C_VEL
LIN {X 0,Y 419.03,Z 611.91,A -85,B 0,C 180,E1 9409.429,E2 9409.429} C_VEL
LIN {X 0,Y 419.027,Z 611.91,A -85,B 0,C 180,E1 9416.21,E2 9416.21} C_VEL
LIN {X 0,Y 419.244,Z 611.91,A -85,B 0,C 180,E1 9421.999,E2 9421.999} C_VEL
LIN {X 0,Y 419.478,Z 611.91,A -85,B 0,C 180,E1 9428.842,E2 9428.842} C_VEL
LIN {X 0,Y 419.691,Z 611.91,A -85,B 0,C 180,E1 9435.373,E2 9435.373} C_VEL
LIN {X 0,Y 419.957,Z 611.91,A -85,B 0,C 180,E1 9441.708,E2 9441.708} C_VEL
LIN {X 0,Y 420.323,Z 611.91,A -85,B 0,C 180,E1 9447.936,E2 9447.936} C_VEL
LIN {X 0,Y 420.117,Z 611.91,A -85,B 0,C 180,E1 9454.133,E2 9454.133} C_VEL
LIN {X 0,Y 419.829,Z 611.91,A -85,B 0,C 180,E1 9460.388,E2 9460.388} C_VEL
LIN {X 0,Y 419.646,Z 611.91,A -85,B 0,C 180,E1 9466.776,E2 9466.776} C_VEL
LIN {X 0,Y 419.388,Z 611.91,A -85,B 0,C 180,E1 9473.398,E2 9473.398} C_VEL
LIN {X 0,Y 419.243,Z 611.91,A -85,B 0,C 180,E1 9480.371,E2 9480.371} C_VEL
LIN {X 0,Y 419.144,Z 611.91,A -85,B 0,C 180,E1 9487.37,E2 9487.37} C_VEL
LIN {X 0,Y 418.882,Z 611.91,A -85,B 0,C 180,E1 9493.702,E2 9493.702} C_VEL
LIN {X 0,Y 418.924,Z 611.91,A -85,B 0,C 180,E1 9499.414,E2 9499.414} C_VEL
LIN {X 0,Y 419.009,Z 611.91,A -85,B 0,C 180,E1 9506.21,E2 9506.21} C_VEL
LIN {X 0,Y 419.245,Z 611.91,A -85,B 0,C 180,E1 9511.996,E2 9511.996} C_VEL
LIN {X 0,Y 419.553,Z 611.91,A -85,B 0,C 180,E1 9518.843,E2 9518.843} C_VEL
LIN {X 0,Y 419.572,Z 611.91,A -85,B 0,C 180,E1 9525.365,E2 9525.365} C_VEL
LIN {X 0,Y 419.944,Z 611.91,A -85,B 0,C 180,E1 9531.705,E2 9531.705} C_VEL
LIN {X 0,Y 420.343,Z 611.91,A -85,B 0,C 180,E1 9537.932,E2 9537.932} C_VEL
LIN {X 0,Y 420.177,Z 611.91,A -85,B 0,C 180,E1 9544.129,E2 9544.129} C_VEL
LIN {X 0,Y 419.844,Z 611.91,A -85,B 0,C 180,E1 9550.384,E2 9550.384} C_VEL
LIN {X 0,Y 419.638,Z 611.91,A -85,B 0,C 180,E1 9556.772,E2 9556.772} C_VEL
LIN {X 0,Y 419.392,Z 611.91,A -85,B 0,C 180,E1 9563.393,E2 9563.393} C_VEL
LIN {X 0,Y 419.176,Z 611.91,A -85,B 0,C 180,E1 9570.371,E2 9570.371} C_VEL
LIN {X 0,Y 419.041,Z 611.91,A -85,B 0,C 180,E1 9577.355,E2 9577.355} C_VEL
LIN {X 0,Y 418.994,Z 611.91,A -85,B 0,C 180,E1 9583.721,E2 9583.721} C_VEL
LIN {X 0,Y 419.154,Z 611.91,A -85,B 0,C 180,E1 9590.491,E2 9590.491} C_VEL
LIN {X 0,Y 419.164,Z 611.91,A -85,B 0,C 180,E1 9591.66,E2 9591.66} C_VEL
LIN {X 0,Y 425.555,Z 625.63,A -85,B 0,C 180,E1 9592.639,E2 9592.639} C_VEL
LIN {X 0,Y 442.548,Z 662.631,A -85,B 0,C 180,E1 9595.185,E2 9595.185} C_VEL
LIN {X 0,Y 444.182,Z 669.138,A -85,B 0,C 180,E1 9595.545,E2 9595.545} C_VEL
LIN {X 0,Y 440.933,Z 705.056,A -85,B 0,C 180,E1 9597.061,E2 9597.061} C_VEL
LIN {X 0,Y 436.872,Z 738.877,A -85,B 0,C 180,E1 9599.245,E2 9599.245} C_VEL
LIN {X 0,Y 432.134,Z 771.938,A -85,B 0,C 180,E1 9602.339,E2 9602.339} C_VEL
LIN {X 0,Y 428.124,Z 798.572,A -85,B 0,C 180,E1 9605.725,E2 9605.725} C_VEL
LIN {X 0,Y 426.047,Z 812.182,A -85,B 0,C 180,E1 9607.917,E2 9607.917} C_VEL
LIN {X 0,Y 420.665,Z 822.629,A -85,B 0,C 180,E1 9609.695,E2 9609.695} C_VEL
LIN {X 0,Y 415.655,Z 832.037,A -85,B 0,C 180,E1 9611.594,E2 9611.594} C_VEL
LIN {X 0,Y 413.738,Z 849.174,A -85,B 0,C 180,E1 9616.452,E2 9616.452} C_VEL
LIN {X 0,Y 412.934,Z 861.098,A -85,B 0,C 180,E1 9621.566,E2 9621.566} C_VEL
LIN {X 0,Y 412.651,Z 866.622,A -85,B 0,C 180,E1 9625.792,E2 9625.792} C_VEL
LIN {X 0,Y 412.635,Z 868.436,A -85,B 0,C 180,E1 9630,E2 9630} C_VEL
LIN {X 0,Y 412.674,Z 866.622,A -85,B 0,C 180,E1 9634.208,E2 9634.208} C_VEL
LIN {X 0,Y 412.978,Z 859.044,A -85,B 0,C 180,E1 9639.496,E2 9639.496} C_VEL
LIN {X 0,Y 413.978,Z 846.686,A -85,B 0,C 180,E1 9644.4,E2 9644.4} C_VEL
LIN {X 0,Y 416.259,Z 827.742,A -85,B 0,C 180,E1 9649.384,E2 9649.384} C_VEL
LIN {X 0,Y 419.63,Z 805.094,A -85,B 0,C 180,E1 9653.666,E2 9653.666} C_VEL
LIN {X 0,Y 424.278,Z 776.401,A -85,B 0,C 180,E1 9657.64,E2 9657.64} C_VEL
LIN {X 0,Y 429.096,Z 744.924,A -85,B 0,C 180,E1 9660.772,E2 9660.772} C_VEL
LIN {X 0,Y 433.587,Z 711.347,A -85,B 0,C 180,E1 9663.156,E2 9663.156} C_VEL
LIN {X 0,Y 437.262,Z 673.353,A -85,B 0,C 180,E1 9664.889,E2 9664.889} C_VEL
LIN {X 0,Y 436.362,Z 666.255,A -85,B 0,C 180,E1 9665.251,E2 9665.251} C_VEL
LIN {X 0,Y 419.86,Z 629.653,A -85,B 0,C 180,E1 9667.867,E2 9667.867} C_VEL
LIN {X 0,Y 411.266,Z 612.632,A -85,B 0,C 180,E1 9669.171,E2 9669.171} C_VEL
LIN {X 0,Y 411.043,Z 611.91,A -85,B 0,C 180,E1 9675.592,E2 9675.592} C_VEL
LIN {X 0,Y 411.028,Z 611.91,A -85,B 0,C 180,E1 9681.236,E2 9681.236} C_VEL
LIN {X 0,Y 411.197,Z 611.91,A -85,B 0,C 180,E1 9687.873,E2 9687.873} C_VEL
LIN {X 0,Y 411.322,Z 611.91,A -85,B 0,C 180,E1 9693.792,E2 9693.792} C_VEL
LIN {X 0,Y 411.571,Z 611.91,A -85,B 0,C 180,E1 9700.67,E2 9700.67} C_VEL
LIN {X 0,Y 411.821,Z 611.91,A -85,B 0,C 180,E1 9707.261,E2 9707.261} C_VEL
LIN {X 0,Y 412.088,Z 611.91,A -85,B 0,C 180,E1 9713.676,E2 9713.676} C_VEL
LIN {X 0,Y 412.368,Z 611.91,A -85,B 0,C 180,E1 9720.004,E2 9720.004} C_VEL
LIN {X 0,Y 412.148,Z 611.91,A -85,B 0,C 180,E1 9726.331,E2 9726.331} C_VEL
LIN {X 0,Y 411.825,Z 611.91,A -85,B 0,C 180,E1 9732.747,E2 9732.747} C_VEL
LIN {X 0,Y 411.61,Z 611.91,A -85,B 0,C 180,E1 9739.336,E2 9739.336} C_VEL
LIN {X 0,Y 411.322,Z 611.91,A -85,B 0,C 180,E1 9746.216,E2 9746.216} C_VEL
LIN {X 0,Y 411.176,Z 611.91,A -85,B 0,C 180,E1 9753.531,E2 9753.531} C_VEL
LIN {X 0,Y 411.068,Z 611.91,A -85,B 0,C 180,E1 9759.333,E2 9759.333} C_VEL
LIN {X 0,Y 411.05,Z 611.91,A -85,B 0,C 180,E1 9765.586,E2 9765.586} C_VEL
LIN {X 0,Y 411.043,Z 611.91,A -85,B 0,C 180,E1 9771.231,E2 9771.231} C_VEL
LIN {X 0,Y 411.137,Z 611.91,A -85,B 0,C 180,E1 9777.89,E2 9777.89} C_VEL
LIN {X 0,Y 411.339,Z 611.91,A -85,B 0,C 180,E1 9783.788,E2 9783.788} C_VEL
LIN {X 0,Y 411.608,Z 611.91,A -85,B 0,C 180,E1 9790.667,E2 9790.667} C_VEL
LIN {X 0,Y 411.831,Z 611.91,A -85,B 0,C 180,E1 9797.257,E2 9797.257} C_VEL
LIN {X 0,Y 412.112,Z 611.91,A -85,B 0,C 180,E1 9803.672,E2 9803.672} C_VEL
LIN {X 0,Y 412.375,Z 611.91,A -85,B 0,C 180,E1 9810,E2 9810} C_VEL
LIN {X 0,Y 412.081,Z 611.91,A -85,B 0,C 180,E1 9816.328,E2 9816.328} C_VEL
LIN {X 0,Y 411.824,Z 611.91,A -85,B 0,C 180,E1 9822.744,E2 9822.744} C_VEL
LIN {X 0,Y 411.609,Z 611.91,A -85,B 0,C 180,E1 9829.333,E2 9829.333} C_VEL
LIN {X 0,Y 411.337,Z 611.91,A -85,B 0,C 180,E1 9836.212,E2 9836.212} C_VEL
LIN {X 0,Y 411.269,Z 611.91,A -85,B 0,C 180,E1 9843.519,E2 9843.519} C_VEL
LIN {X 0,Y 411.067,Z 611.91,A -85,B 0,C 180,E1 9849.33,E2 9849.33} C_VEL
LIN {X 0,Y 410.887,Z 611.91,A -85,B 0,C 180,E1 9855.56,E2 9855.56} C_VEL
LIN {X 0,Y 410.963,Z 611.91,A -85,B 0,C 180,E1 9861.219,E2 9861.219} C_VEL
LIN {X 0,Y 411.128,Z 611.91,A -85,B 0,C 180,E1 9867.889,E2 9867.889} C_VEL
LIN {X 0,Y 411.348,Z 611.91,A -85,B 0,C 180,E1 9873.785,E2 9873.785} C_VEL
LIN {X 0,Y 411.68,Z 611.91,A -85,B 0,C 180,E1 9880.667,E2 9880.667} C_VEL
LIN {X 0,Y 411.701,Z 611.91,A -85,B 0,C 180,E1 9887.249,E2 9887.249} C_VEL
LIN {X 0,Y 412.148,Z 611.91,A -85,B 0,C 180,E1 9893.669,E2 9893.669} C_VEL
LIN {X 0,Y 412.444,Z 611.91,A -85,B 0,C 180,E1 9899.996,E2 9899.996} C_VEL
LIN {X 0,Y 412.086,Z 611.91,A -85,B 0,C 180,E1 9906.324,E2 9906.324} C_VEL
LIN {X 0,Y 411.831,Z 611.91,A -85,B 0,C 180,E1 9912.739,E2 9912.739} C_VEL
LIN {X 0,Y 411.607,Z 611.91,A -85,B 0,C 180,E1 9919.328,E2 9919.328} C_VEL
LIN {X 0,Y 411.344,Z 611.91,A -85,B 0,C 180,E1 9926.206,E2 9926.206} C_VEL
LIN {X 0,Y 411.159,Z 611.91,A -85,B 0,C 180,E1 9933.523,E2 9933.523} C_VEL
LIN {X 0,Y 411.018,Z 611.91,A -85,B 0,C 180,E1 9939.324,E2 9939.324} C_VEL
LIN {X 0,Y 411.068,Z 611.91,A -85,B 0,C 180,E1 9945.588,E2 9945.588} C_VEL
LIN {X 0,Y 411.28,Z 612.526,A -85,B 0,C 180,E1 9950.829,E2 9950.829} C_VEL
LIN {X 0,Y 433.592,Z 659.034,A -85,B 0,C 180,E1 9954.245,E2 9954.245} C_VEL
LIN {X 0,Y 437.487,Z 670.846,A -85,B 0,C 180,E1 9955.022,E2 9955.022} C_VEL
LIN {X 0,Y 433.799,Z 708.964,A -85,B 0,C 180,E1 9956.712,E2 9956.712} C_VEL
LIN {X 0,Y 429.505,Z 741.865,A -85,B 0,C 180,E1 9958.966,E2 9958.966} C_VEL
LIN {X 0,Y 424.486,Z 775.288,A -85,B 0,C 180,E1 9962.231,E2 9962.231} C_VEL
LIN {X 0,Y 419.878,Z 803.403,A -85,B 0,C 180,E1 9966.067,E2 9966.067} C_VEL
LIN {X 0,Y 416.423,Z 826.565,A -85,B 0,C 180,E1 9970.347,E2 9970.347} C_VEL
LIN {X 0,Y 415.655,Z 832.037,A -85,B 0,C 180,E1 9971.594,E2 9971.594} C_VEL
LIN {X 0,Y 412.495,Z 838.525,A -85,B 0,C 180,E1 9973.112,E2 9973.112} C_VEL
LIN {X 0,Y 406.236,Z 846.937,A -85,B 0,C 180,E1 9975.475,E2 9975.475} C_VEL
LIN {X 0,Y 406.041,Z 847.751,A -85,B 0,C 180,E1 9975.761,E2 9975.761} C_VEL
LIN {X 0,Y 405.065,Z 859.835,A -85,B 0,C 180,E1 9980.859,E2 9980.859} C_VEL
LIN {X 0,Y 404.768,Z 866.388,A -85,B 0,C 180,E1 9985.71,E2 9985.71} C_VEL
LIN {X 0,Y 404.738,Z 868.203,A -85,B 0,C 180,E1 9990,E2 9990} C_VEL
LIN {X 0,Y 404.789,Z 866.389,A -85,B 0,C 180,E1 9994.29,E2 9994.29} C_VEL
LIN {X 0,Y 405.115,Z 858.808,A -85,B 0,C 180,E1 9999.682,E2 9999.682} C_VEL
LIN {X 0,Y 406.163,Z 846.817,A -85,B 0,C 180,E1 10004.567,E2 10004.567} C_VEL
LIN {X 0,Y 408.624,Z 827.502,A -85,B 0,C 180,E1 10009.761,E2 10009.761} C_VEL
LIN {X 0,Y 412.228,Z 804.855,A -85,B 0,C 180,E1 10014.117,E2 10014.117} C_VEL
LIN {X 0,Y 417.105,Z 776.161,A -85,B 0,C 180,E1 10018.157,E2 10018.157} C_VEL
LIN {X 0,Y 422.238,Z 744.688,A -85,B 0,C 180,E1 10021.328,E2 10021.328} C_VEL
LIN {X 0,Y 426.926,Z 711.106,A -85,B 0,C 180,E1 10023.742,E2 10023.742} C_VEL
LIN {X 0,Y 430.813,Z 672.93,A -85,B 0,C 180,E1 10025.498,E2 10025.498} C_VEL
LIN {X 0,Y 419.012,Z 643.399,A -85,B 0,C 180,E1 10027.646,E2 10027.646} C_VEL
LIN {X 0,Y 403.334,Z 613.21,A -85,B 0,C 180,E1 10030.075,E2 10030.075} C_VEL
LIN {X 0,Y 403.2,Z 611.91,A -85,B 0,C 180,E1 10030.25,E2 10030.25} C_VEL
LIN {X 0,Y 403.111,Z 611.91,A -85,B 0,C 180,E1 10037.47,E2 10037.47} C_VEL
LIN {X 0,Y 403.108,Z 611.91,A -85,B 0,C 180,E1 10043.068,E2 10043.068} C_VEL
LIN {X 0,Y 403.283,Z 611.91,A -85,B 0,C 180,E1 10049.711,E2 10049.711} C_VEL
LIN {X 0,Y 403.422,Z 611.91,A -85,B 0,C 180,E1 10055.622,E2 10055.622} C_VEL
LIN {X 0,Y 403.729,Z 611.91,A -85,B 0,C 180,E1 10062.546,E2 10062.546} C_VEL
LIN {X 0,Y 403.973,Z 611.91,A -85,B 0,C 180,E1 10069.204,E2 10069.204} C_VEL
LIN {X 0,Y 404.284,Z 611.91,A -85,B 0,C 180,E1 10075.709,E2 10075.709} C_VEL
LIN {X 0,Y 404.533,Z 611.91,A -85,B 0,C 180,E1 10082.149,E2 10082.149} C_VEL
LIN {X 0,Y 404.106,Z 611.91,A -85,B 0,C 180,E1 10088.623,E2 10088.623} C_VEL
LIN {X 0,Y 403.81,Z 611.91,A -85,B 0,C 180,E1 10095.219,E2 10095.219} C_VEL
LIN {X 0,Y 403.569,Z 611.91,A -85,B 0,C 180,E1 10102.038,E2 10102.038} C_VEL
LIN {X 0,Y 403.295,Z 611.91,A -85,B 0,C 180,E1 10109.216,E2 10109.216} C_VEL
LIN {X 0,Y 403.208,Z 611.91,A -85,B 0,C 180,E1 10114.299,E2 10114.299} C_VEL
LIN {X 0,Y 403.119,Z 611.91,A -85,B 0,C 180,E1 10121.308,E2 10121.308} C_VEL
LIN {X 0,Y 403.141,Z 611.91,A -85,B 0,C 180,E1 10127.467,E2 10127.467} C_VEL
LIN {X 0,Y 403.086,Z 611.91,A -85,B 0,C 180,E1 10133.06,E2 10133.06} C_VEL
LIN {X 0,Y 403.249,Z 611.91,A -85,B 0,C 180,E1 10139.723,E2 10139.723} C_VEL
LIN {X 0,Y 403.46,Z 611.91,A -85,B 0,C 180,E1 10145.62,E2 10145.62} C_VEL
LIN {X 0,Y 403.722,Z 611.91,A -85,B 0,C 180,E1 10152.541,E2 10152.541} C_VEL
LIN {X 0,Y 403.945,Z 611.91,A -85,B 0,C 180,E1 10159.198,E2 10159.198} C_VEL
LIN {X 0,Y 404.227,Z 611.91,A -85,B 0,C 180,E1 10165.704,E2 10165.704} C_VEL
LIN {X 0,Y 404.401,Z 611.91,A -85,B 0,C 180,E1 10172.146,E2 10172.146} C_VEL
LIN {X 0,Y 404.104,Z 611.91,A -85,B 0,C 180,E1 10178.619,E2 10178.619} C_VEL
LIN {X 0,Y 403.819,Z 611.91,A -85,B 0,C 180,E1 10185.216,E2 10185.216} C_VEL
LIN {X 0,Y 403.58,Z 611.91,A -85,B 0,C 180,E1 10192.034,E2 10192.034} C_VEL
LIN {X 0,Y 403.345,Z 611.91,A -85,B 0,C 180,E1 10199.208,E2 10199.208} C_VEL
LIN {X 0,Y 403.304,Z 611.91,A -85,B 0,C 180,E1 10204.316,E2 10204.316} C_VEL
LIN {X 0,Y 403.065,Z 611.91,A -85,B 0,C 180,E1 10211.296,E2 10211.296} C_VEL
LIN {X 0,Y 402.99,Z 611.91,A -85,B 0,C 180,E1 10217.444,E2 10217.444} C_VEL
LIN {X 0,Y 403.041,Z 611.91,A -85,B 0,C 180,E1 10223.052,E2 10223.052} C_VEL
LIN {X 0,Y 403.245,Z 611.91,A -85,B 0,C 180,E1 10229.72,E2 10229.72} C_VEL
LIN {X 0,Y 403.484,Z 611.91,A -85,B 0,C 180,E1 10235.618,E2 10235.618} C_VEL
LIN {X 0,Y 403.732,Z 611.91,A -85,B 0,C 180,E1 10242.538,E2 10242.538} C_VEL
LIN {X 0,Y 403.865,Z 611.91,A -85,B 0,C 180,E1 10249.193,E2 10249.193} C_VEL
LIN {X 0,Y 404.261,Z 611.91,A -85,B 0,C 180,E1 10255.701,E2 10255.701} C_VEL
LIN {X 0,Y 404.408,Z 611.91,A -85,B 0,C 180,E1 10262.142,E2 10262.142} C_VEL
LIN {X 0,Y 404.103,Z 611.91,A -85,B 0,C 180,E1 10268.615,E2 10268.615} C_VEL
LIN {X 0,Y 403.808,Z 611.91,A -85,B 0,C 180,E1 10275.211,E2 10275.211} C_VEL
LIN {X 0,Y 403.582,Z 611.91,A -85,B 0,C 180,E1 10282.029,E2 10282.029} C_VEL
LIN {X 0,Y 403.297,Z 611.91,A -85,B 0,C 180,E1 10289.206,E2 10289.206} C_VEL
LIN {X 0,Y 403.176,Z 611.91,A -85,B 0,C 180,E1 10294.293,E2 10294.293} C_VEL
LIN {X 0,Y 403.081,Z 611.91,A -85,B 0,C 180,E1 10301.302,E2 10301.302} C_VEL
LIN {X 0,Y 403.174,Z 611.91,A -85,B 0,C 180,E1 10307.471,E2 10307.471} C_VEL
LIN {X 0,Y 403.235,Z 611.91,A -85,B 0,C 180,E1 10309.879,E2 10309.879} C_VEL
LIN {X 0,Y 407.593,Z 621.518,A -85,B 0,C 180,E1 10310.609,E2 10310.609} C_VEL
LIN {X 0,Y 425.707,Z 658.318,A -85,B 0,C 180,E1 10313.462,E2 10313.462} C_VEL
LIN {X 0,Y 430.817,Z 672.905,A -85,B 0,C 180,E1 10314.501,E2 10314.501} C_VEL
LIN {X 0,Y 426.997,Z 710.16,A -85,B 0,C 180,E1 10316.203,E2 10316.203} C_VEL
LIN {X 0,Y 422.157,Z 744.685,A -85,B 0,C 180,E1 10318.665,E2 10318.665} C_VEL
LIN {X 0,Y 417.146,Z 776.163,A -85,B 0,C 180,E1 10321.846,E2 10321.846} C_VEL
LIN {X 0,Y 412.224,Z 804.855,A -85,B 0,C 180,E1 10325.883,E2 10325.883} C_VEL
LIN {X 0,Y 408.607,Z 827.502,A -85,B 0,C 180,E1 10330.238,E2 10330.238} C_VEL
LIN {X 0,Y 406.166,Z 846.807,A -85,B 0,C 180,E1 10335.43,E2 10335.43} C_VEL
LIN {X 0,Y 406.041,Z 847.751,A -85,B 0,C 180,E1 10335.761,E2 10335.761} C_VEL
LIN {X 0,Y 401.517,Z 853.917,A -85,B 0,C 180,E1 10338.003,E2 10338.003} C_VEL
LIN {X 0,Y 397.229,Z 858.975,A -85,B 0,C 180,E1 10340.341,E2 10340.341} C_VEL
LIN {X 0,Y 396.869,Z 866.154,A -85,B 0,C 180,E1 10345.624,E2 10345.624} C_VEL
LIN {X 0,Y 396.841,Z 867.969,A -85,B 0,C 180,E1 10350,E2 10350} C_VEL
LIN {X 0,Y 396.889,Z 866.154,A -85,B 0,C 180,E1 10354.376,E2 10354.376} C_VEL
LIN {X 0,Y 397.255,Z 858.572,A -85,B 0,C 180,E1 10359.876,E2 10359.876} C_VEL
LIN {X 0,Y 398.385,Z 846.284,A -85,B 0,C 180,E1 10364.954,E2 10364.954} C_VEL
LIN {X 0,Y 401.014,Z 827.263,A -85,B 0,C 180,E1 10370.153,E2 10370.153} C_VEL
LIN {X 0,Y 404.867,Z 804.616,A -85,B 0,C 180,E1 10374.584,E2 10374.584} C_VEL
LIN {X 0,Y 409.963,Z 775.921,A -85,B 0,C 180,E1 10378.693,E2 10378.693} C_VEL
LIN {X 0,Y 415.393,Z 744.45,A -85,B 0,C 180,E1 10381.905,E2 10381.905} C_VEL
LIN {X 0,Y 420.274,Z 711.073,A -85,B 0,C 180,E1 10384.336,E2 10384.336} C_VEL
LIN {X 0,Y 423.711,Z 672.858,A -85,B 0,C 180,E1 10386.178,E2 10386.178} C_VEL
LIN {X 0,Y 409.225,Z 639.079,A -85,B 0,C 180,E1 10388.817,E2 10388.817} C_VEL
LIN {X 0,Y 395.306,Z 612.804,A -85,B 0,C 180,E1 10391.063,E2 10391.063} C_VEL
LIN {X 0,Y 395.256,Z 611.91,A -85,B 0,C 180,E1 10391.265,E2 10391.265} C_VEL
LIN {X 0,Y 395.168,Z 611.91,A -85,B 0,C 180,E1 10396.716,E2 10396.716} C_VEL
LIN {X 0,Y 395.178,Z 611.91,A -85,B 0,C 180,E1 10403.57,E2 10403.57} C_VEL
LIN {X 0,Y 395.406,Z 611.91,A -85,B 0,C 180,E1 10410.152,E2 10410.152} C_VEL
LIN {X 0,Y 395.55,Z 611.91,A -85,B 0,C 180,E1 10417.5,E2 10417.5} C_VEL
LIN {X 0,Y 395.854,Z 611.91,A -85,B 0,C 180,E1 10424.475,E2 10424.475} C_VEL
LIN {X 0,Y 396.178,Z 611.91,A -85,B 0,C 180,E1 10431.211,E2 10431.211} C_VEL
LIN {X 0,Y 396.485,Z 611.91,A -85,B 0,C 180,E1 10437.816,E2 10437.816} C_VEL
LIN {X 0,Y 396.618,Z 611.91,A -85,B 0,C 180,E1 10442.192,E2 10442.192} C_VEL
LIN {X 0,Y 396.177,Z 611.91,A -85,B 0,C 180,E1 10448.797,E2 10448.797} C_VEL
LIN {X 0,Y 395.864,Z 611.91,A -85,B 0,C 180,E1 10455.533,E2 10455.533} C_VEL
LIN {X 0,Y 395.591,Z 611.91,A -85,B 0,C 180,E1 10462.506,E2 10462.506} C_VEL
LIN {X 0,Y 395.374,Z 611.91,A -85,B 0,C 180,E1 10469.859,E2 10469.859} C_VEL
LIN {X 0,Y 395.195,Z 611.91,A -85,B 0,C 180,E1 10476.434,E2 10476.434} C_VEL
LIN {X 0,Y 395.19,Z 611.91,A -85,B 0,C 180,E1 10483.287,E2 10483.287} C_VEL
LIN {X 0,Y 395.206,Z 611.91,A -85,B 0,C 180,E1 10490.018,E2 10490.018} C_VEL
LIN {X 0,Y 395.241,Z 611.91,A -85,B 0,C 180,E1 10497.568,E2 10497.568} C_VEL
LIN {X 0,Y 395.414,Z 611.91,A -85,B 0,C 180,E1 10502.646,E2 10502.646} C_VEL
LIN {X 0,Y 395.727,Z 611.91,A -85,B 0,C 180,E1 10509.858,E2 10509.858} C_VEL
LIN {X 0,Y 395.972,Z 611.91,A -85,B 0,C 180,E1 10516.737,E2 10516.737} C_VEL
LIN {X 0,Y 396.277,Z 611.91,A -85,B 0,C 180,E1 10523.418,E2 10523.418} C_VEL
LIN {X 0,Y 396.579,Z 611.91,A -85,B 0,C 180,E1 10530,E2 10530} C_VEL
LIN {X 0,Y 396.277,Z 611.91,A -85,B 0,C 180,E1 10536.582,E2 10536.582} C_VEL
LIN {X 0,Y 395.972,Z 611.91,A -85,B 0,C 180,E1 10543.263,E2 10543.263} C_VEL
LIN {X 0,Y 395.729,Z 611.91,A -85,B 0,C 180,E1 10550.141,E2 10550.141} C_VEL
LIN {X 0,Y 395.426,Z 611.91,A -85,B 0,C 180,E1 10557.353,E2 10557.353} C_VEL
LIN {X 0,Y 395.357,Z 611.91,A -85,B 0,C 180,E1 10562.59,E2 10562.59} C_VEL
LIN {X 0,Y 395.251,Z 611.91,A -85,B 0,C 180,E1 10567.799,E2 10567.799} C_VEL
LIN {X 0,Y 395.091,Z 611.91,A -85,B 0,C 180,E1 10573.613,E2 10573.613} C_VEL
LIN {X 0,Y 395.091,Z 611.91,A -85,B 0,C 180,E1 10580.035,E2 10580.035} C_VEL
LIN {X 0,Y 395.224,Z 611.91,A -85,B 0,C 180,E1 10587.436,E2 10587.436} C_VEL
LIN {X 0,Y 395.417,Z 611.91,A -85,B 0,C 180,E1 10592.643,E2 10592.643} C_VEL
LIN {X 0,Y 395.795,Z 611.91,A -85,B 0,C 180,E1 10599.859,E2 10599.859} C_VEL
LIN {X 0,Y 395.846,Z 611.91,A -85,B 0,C 180,E1 10606.729,E2 10606.729} C_VEL
LIN {X 0,Y 396.319,Z 611.91,A -85,B 0,C 180,E1 10613.415,E2 10613.415} C_VEL
LIN {X 0,Y 396.641,Z 611.91,A -85,B 0,C 180,E1 10619.996,E2 10619.996} C_VEL
LIN {X 0,Y 396.262,Z 611.91,A -85,B 0,C 180,E1 10626.578,E2 10626.578} C_VEL
LIN {X 0,Y 395.96,Z 611.91,A -85,B 0,C 180,E1 10633.259,E2 10633.259} C_VEL
LIN {X 0,Y 395.728,Z 611.91,A -85,B 0,C 180,E1 10640.136,E2 10640.136} C_VEL
LIN {X 0,Y 395.41,Z 611.91,A -85,B 0,C 180,E1 10647.348,E2 10647.348} C_VEL
LIN {X 0,Y 395.26,Z 611.91,A -85,B 0,C 180,E1 10652.572,E2 10652.572} C_VEL
LIN {X 0,Y 395.176,Z 611.91,A -85,B 0,C 180,E1 10659.98,E2 10659.98} C_VEL
LIN {X 0,Y 395.227,Z 611.91,A -85,B 0,C 180,E1 10666.699,E2 10666.699} C_VEL
LIN {X 0,Y 395.291,Z 611.91,A -85,B 0,C 180,E1 10668.873,E2 10668.873} C_VEL
LIN {X 0,Y 399.92,Z 621.895,A -85,B 0,C 180,E1 10669.716,E2 10669.716} C_VEL
LIN {X 0,Y 418.413,Z 658.875,A -85,B 0,C 180,E1 10672.748,E2 10672.748} C_VEL
LIN {X 0,Y 424.226,Z 674.56,A -85,B 0,C 180,E1 10673.95,E2 10673.95} C_VEL
LIN {X 0,Y 420.158,Z 711.745,A -85,B 0,C 180,E1 10675.701,E2 10675.701} C_VEL
LIN {X 0,Y 414.837,Z 747.507,A -85,B 0,C 180,E1 10678.355,E2 10678.355} C_VEL
LIN {X 0,Y 409.71,Z 777.849,A -85,B 0,C 180,E1 10681.56,E2 10681.56} C_VEL
LIN {X 0,Y 404.556,Z 806.306,A -85,B 0,C 180,E1 10685.69,E2 10685.69} C_VEL
LIN {X 0,Y 400.617,Z 829.577,A -85,B 0,C 180,E1 10690.393,E2 10690.393} C_VEL
LIN {X 0,Y 398.233,Z 847.603,A -85,B 0,C 180,E1 10695.509,E2 10695.509} C_VEL
LIN {X 0,Y 397.229,Z 858.975,A -85,B 0,C 180,E1 10700.341,E2 10700.341} C_VEL
LIN {X 0,Y 394.543,Z 862.064,A -85,B 0,C 180,E1 10702.149,E2 10702.149} C_VEL
LIN {X 0,Y 389.086,Z 865.299,A -85,B 0,C 180,E1 10704.907,E2 10704.907} C_VEL
LIN {X 0,Y 388.98,Z 865.613,A -85,B 0,C 180,E1 10705.228,E2 10705.228} C_VEL
LIN {X 0,Y 388.965,Z 867.737,A -85,B 0,C 180,E1 10710,E2 10710} C_VEL
LIN {X 0,Y 388.991,Z 865.92,A -85,B 0,C 180,E1 10714.465,E2 10714.465} C_VEL
LIN {X 0,Y 389.336,Z 859.364,A -85,B 0,C 180,E1 10719.513,E2 10719.513} C_VEL
LIN {X 0,Y 390.428,Z 847.526,A -85,B 0,C 180,E1 10724.727,E2 10724.727} C_VEL
LIN {X 0,Y 392.812,Z 830.504,A -85,B 0,C 180,E1 10729.722,E2 10729.722} C_VEL
LIN {X 0,Y 396.978,Z 807.275,A -85,B 0,C 180,E1 10734.582,E2 10734.582} C_VEL
LIN {X 0,Y 402.346,Z 778.879,A -85,B 0,C 180,E1 10738.825,E2 10738.825} C_VEL
LIN {X 0,Y 407.817,Z 748.8,A -85,B 0,C 180,E1 10742.098,E2 10742.098} C_VEL
LIN {X 0,Y 413.224,Z 714.198,A -85,B 0,C 180,E1 10744.745,E2 10744.745} C_VEL
LIN {X 0,Y 417.387,Z 678.314,A -85,B 0,C 180,E1 10746.55,E2 10746.55} C_VEL
LIN {X 0,Y 411.435,Z 660.398,A -85,B 0,C 180,E1 10747.928,E2 10747.928} C_VEL
LIN {X 0,Y 394.212,Z 625.826,A -85,B 0,C 180,E1 10750.894,E2 10750.894} C_VEL
LIN {X 0,Y 387.439,Z 613.318,A -85,B 0,C 180,E1 10752.064,E2 10752.064} C_VEL
LIN {X 0,Y 387.291,Z 611.91,A -85,B 0,C 180,E1 10752.192,E2 10752.192} C_VEL
LIN {X 0,Y 387.167,Z 611.91,A -85,B 0,C 180,E1 10758.34,E2 10758.34} C_VEL
LIN {X 0,Y 387.321,Z 611.91,A -85,B 0,C 180,E1 10765.175,E2 10765.175} C_VEL
LIN {X 0,Y 387.508,Z 611.91,A -85,B 0,C 180,E1 10772.046,E2 10772.046} C_VEL
LIN {X 0,Y 387.753,Z 611.91,A -85,B 0,C 180,E1 10779.574,E2 10779.574} C_VEL
LIN {X 0,Y 388.029,Z 611.91,A -85,B 0,C 180,E1 10786.465,E2 10786.465} C_VEL
LIN {X 0,Y 388.34,Z 611.91,A -85,B 0,C 180,E1 10793.287,E2 10793.287} C_VEL
LIN {X 0,Y 388.679,Z 611.91,A -85,B 0,C 180,E1 10800.004,E2 10800.004} C_VEL
LIN {X 0,Y 388.419,Z 611.91,A -85,B 0,C 180,E1 10806.719,E2 10806.719} C_VEL
LIN {X 0,Y 388.04,Z 611.91,A -85,B 0,C 180,E1 10813.543,E2 10813.543} C_VEL
LIN {X 0,Y 387.754,Z 611.91,A -85,B 0,C 180,E1 10820.578,E2 10820.578} C_VEL
LIN {X 0,Y 387.491,Z 611.91,A -85,B 0,C 180,E1 10827.965,E2 10827.965} C_VEL
LIN {X 0,Y 387.281,Z 611.91,A -85,B 0,C 180,E1 10835.906,E2 10835.906} C_VEL
LIN {X 0,Y 387.193,Z 611.91,A -85,B 0,C 180,E1 10842.016,E2 10842.016} C_VEL
LIN {X 0,Y 387.194,Z 611.91,A -85,B 0,C 180,E1 10848.336,E2 10848.336} C_VEL
LIN {X 0,Y 387.219,Z 611.91,A -85,B 0,C 180,E1 10855.2,E2 10855.2} C_VEL
LIN {X 0,Y 387.505,Z 611.91,A -85,B 0,C 180,E1 10862.04,E2 10862.04} C_VEL
LIN {X 0,Y 387.781,Z 611.91,A -85,B 0,C 180,E1 10869.568,E2 10869.568} C_VEL
LIN {X 0,Y 388.043,Z 611.91,A -85,B 0,C 180,E1 10876.461,E2 10876.461} C_VEL
LIN {X 0,Y 388.353,Z 611.91,A -85,B 0,C 180,E1 10883.283,E2 10883.283} C_VEL
LIN {X 0,Y 388.687,Z 611.91,A -85,B 0,C 180,E1 10890,E2 10890} C_VEL
LIN {X 0,Y 388.353,Z 611.91,A -85,B 0,C 180,E1 10896.717,E2 10896.717} C_VEL
LIN {X 0,Y 388.045,Z 611.91,A -85,B 0,C 180,E1 10903.539,E2 10903.539} C_VEL
LIN {X 0,Y 387.757,Z 611.91,A -85,B 0,C 180,E1 10910.574,E2 10910.574} C_VEL
LIN {X 0,Y 387.524,Z 611.91,A -85,B 0,C 180,E1 10917.959,E2 10917.959} C_VEL
LIN {X 0,Y 387.396,Z 611.91,A -85,B 0,C 180,E1 10924.837,E2 10924.837} C_VEL
LIN {X 0,Y 387.132,Z 611.91,A -85,B 0,C 180,E1 10932.002,E2 10932.002} C_VEL
LIN {X 0,Y 387.068,Z 611.91,A -85,B 0,C 180,E1 10938.316,E2 10938.316} C_VEL
LIN {X 0,Y 387.204,Z 611.91,A -85,B 0,C 180,E1 10945.2,E2 10945.2} C_VEL
LIN {X 0,Y 387.507,Z 611.91,A -85,B 0,C 180,E1 10952.036,E2 10952.036} C_VEL
LIN {X 0,Y 387.844,Z 611.91,A -85,B 0,C 180,E1 10959.538,E2 10959.538} C_VEL
LIN {X 0,Y 387.92,Z 611.91,A -85,B 0,C 180,E1 10966.453,E2 10966.453} C_VEL
LIN {X 0,Y 388.417,Z 611.91,A -85,B 0,C 180,E1 10973.281,E2 10973.281} C_VEL
LIN {X 0,Y 388.745,Z 611.91,A -85,B 0,C 180,E1 10979.996,E2 10979.996} C_VEL
LIN {X 0,Y 388.339,Z 611.91,A -85,B 0,C 180,E1 10986.713,E2 10986.713} C_VEL
LIN {X 0,Y 388.032,Z 611.91,A -85,B 0,C 180,E1 10993.535,E2 10993.535} C_VEL
LIN {X 0,Y 387.786,Z 611.91,A -85,B 0,C 180,E1 11000.567,E2 11000.567} C_VEL
LIN {X 0,Y 387.497,Z 611.91,A -85,B 0,C 180,E1 11007.955,E2 11007.955} C_VEL
LIN {X 0,Y 387.277,Z 611.91,A -85,B 0,C 180,E1 11014.816,E2 11014.816} C_VEL
LIN {X 0,Y 387.164,Z 611.91,A -85,B 0,C 180,E1 11022.011,E2 11022.011} C_VEL
LIN {X 0,Y 387.294,Z 611.96,A -85,B 0,C 180,E1 11027.883,E2 11027.883} C_VEL
LIN {X 0,Y 389.895,Z 617.742,A -85,B 0,C 180,E1 11028.365,E2 11028.365} C_VEL
LIN {X 0,Y 410.312,Z 657.535,A -85,B 0,C 180,E1 11031.844,E2 11031.844} C_VEL
LIN {X 0,Y 417.438,Z 678.361,A -85,B 0,C 180,E1 11033.457,E2 11033.457} C_VEL
LIN {X 0,Y 413.122,Z 714.445,A -85,B 0,C 180,E1 11035.265,E2 11035.265} C_VEL
LIN {X 0,Y 407.538,Z 750.326,A -85,B 0,C 180,E1 11038.035,E2 11038.035} C_VEL
LIN {X 0,Y 401.705,Z 782.071,A -85,B 0,C 180,E1 11041.586,E2 11041.586} C_VEL
LIN {X 0,Y 396.743,Z 808.361,A -85,B 0,C 180,E1 11045.619,E2 11045.619} C_VEL
LIN {X 0,Y 392.579,Z 832.009,A -85,B 0,C 180,E1 11050.641,E2 11050.641} C_VEL
LIN {X 0,Y 390.247,Z 849.176,A -85,B 0,C 180,E1 11055.889,E2 11055.889} C_VEL
LIN {X 0,Y 389.258,Z 860.39,A -85,B 0,C 180,E1 11061.049,E2 11061.049} C_VEL
LIN {X 0,Y 388.98,Z 865.613,A -85,B 0,C 180,E1 11065.228,E2 11065.228} C_VEL
LIN {X 0,Y 386.469,Z 867.034,A -85,B 0,C 180,E1 11067.115,E2 11067.115} C_VEL
LIN {X 0,Y 381.03,Z 867.442,A -85,B 0,C 180,E1 11070.305,E2 11070.305} C_VEL
LIN {X 0,Y 381.174,Z 864.568,A -85,B 0,C 180,E1 11075.699,E2 11075.699} C_VEL
LIN {X 0,Y 381.608,Z 857.072,A -85,B 0,C 180,E1 11080.863,E2 11080.863} C_VEL
LIN {X 0,Y 383.015,Z 844.307,A -85,B 0,C 180,E1 11086.064,E2 11086.064} C_VEL
LIN {X 0,Y 386.028,Z 825.607,A -85,B 0,C 180,E1 11091.272,E2 11091.272} C_VEL
LIN {X 0,Y 390.45,Z 802.565,A -85,B 0,C 180,E1 11095.843,E2 11095.843} C_VEL
LIN {X 0,Y 396.175,Z 774.042,A -85,B 0,C 180,E1 11099.986,E2 11099.986} C_VEL
LIN {X 0,Y 402.339,Z 740.916,A -85,B 0,C 180,E1 11103.392,E2 11103.392} C_VEL
LIN {X 0,Y 407.533,Z 708.233,A -85,B 0,C 180,E1 11105.734,E2 11105.734} C_VEL
LIN {X 0,Y 410.416,Z 677.471,A -85,B 0,C 180,E1 11107.303,E2 11107.303} C_VEL
LIN {X 0,Y 396.594,Z 644.685,A -85,B 0,C 180,E1 11110.127,E2 11110.127} C_VEL
LIN {X 0,Y 379.432,Z 612.542,A -85,B 0,C 180,E1 11113.177,E2 11113.177} C_VEL
LIN {X 0,Y 379.185,Z 611.91,A -85,B 0,C 180,E1 11120.3,E2 11120.3} C_VEL
LIN {X 0,Y 379.447,Z 611.91,A -85,B 0,C 180,E1 11126.922,E2 11126.922} C_VEL
LIN {X 0,Y 379.6,Z 611.91,A -85,B 0,C 180,E1 11133.982,E2 11133.982} C_VEL
LIN {X 0,Y 379.886,Z 611.91,A -85,B 0,C 180,E1 11141.412,E2 11141.412} C_VEL
LIN {X 0,Y 380.177,Z 611.91,A -85,B 0,C 180,E1 11148.519,E2 11148.519} C_VEL
LIN {X 0,Y 380.549,Z 611.91,A -85,B 0,C 180,E1 11155.44,E2 11155.44} C_VEL
LIN {X 0,Y 380.808,Z 611.91,A -85,B 0,C 180,E1 11162.283,E2 11162.283} C_VEL
LIN {X 0,Y 380.315,Z 611.91,A -85,B 0,C 180,E1 11169.167,E2 11169.167} C_VEL
LIN {X 0,Y 379.994,Z 611.91,A -85,B 0,C 180,E1 11176.199,E2 11176.199} C_VEL
LIN {X 0,Y 379.668,Z 611.91,A -85,B 0,C 180,E1 11183.506,E2 11183.506} C_VEL
LIN {X 0,Y 379.402,Z 611.91,A -85,B 0,C 180,E1 11191.254,E2 11191.254} C_VEL
LIN {X 0,Y 379.273,Z 611.91,A -85,B 0,C 180,E1 11197.023,E2 11197.023} C_VEL
LIN {X 0,Y 379.205,Z 611.91,A -85,B 0,C 180,E1 11204.054,E2 11204.054} C_VEL
LIN {X 0,Y 379.202,Z 611.91,A -85,B 0,C 180,E1 11210.295,E2 11210.295} C_VEL
LIN {X 0,Y 379.357,Z 611.91,A -85,B 0,C 180,E1 11216.947,E2 11216.947} C_VEL
LIN {X 0,Y 379.622,Z 611.91,A -85,B 0,C 180,E1 11223.978,E2 11223.978} C_VEL
LIN {X 0,Y 379.9,Z 611.91,A -85,B 0,C 180,E1 11231.408,E2 11231.408} C_VEL
LIN {X 0,Y 380.162,Z 611.91,A -85,B 0,C 180,E1 11238.514,E2 11238.514} C_VEL
LIN {X 0,Y 380.506,Z 611.91,A -85,B 0,C 180,E1 11245.435,E2 11245.435} C_VEL
LIN {X 0,Y 380.786,Z 611.91,A -85,B 0,C 180,E1 11250,E2 11250} C_VEL
LIN {X 0,Y 380.441,Z 611.91,A -85,B 0,C 180,E1 11256.857,E2 11256.857} C_VEL
LIN {X 0,Y 380.099,Z 611.91,A -85,B 0,C 180,E1 11263.827,E2 11263.827} C_VEL
LIN {X 0,Y 379.784,Z 611.91,A -85,B 0,C 180,E1 11271.026,E2 11271.026} C_VEL
LIN {X 0,Y 379.524,Z 611.91,A -85,B 0,C 180,E1 11278.635,E2 11278.635} C_VEL
LIN {X 0,Y 379.467,Z 611.91,A -85,B 0,C 180,E1 11283.959,E2 11283.959} C_VEL
LIN {X 0,Y 379.18,Z 611.91,A -85,B 0,C 180,E1 11290.65,E2 11290.65} C_VEL
LIN {X 0,Y 379.083,Z 611.91,A -85,B 0,C 180,E1 11297.233,E2 11297.233} C_VEL
LIN {X 0,Y 379.198,Z 611.91,A -85,B 0,C 180,E1 11303.204,E2 11303.204} C_VEL
LIN {X 0,Y 379.381,Z 611.91,A -85,B 0,C 180,E1 11308.744,E2 11308.744} C_VEL
LIN {X 0,Y 379.731,Z 611.91,A -85,B 0,C 180,E1 11316.498,E2 11316.498} C_VEL
LIN {X 0,Y 379.94,Z 611.91,A -85,B 0,C 180,E1 11323.799,E2 11323.799} C_VEL
LIN {X 0,Y 380.288,Z 611.91,A -85,B 0,C 180,E1 11331.545,E2 11331.545} C_VEL
LIN {X 0,Y 380.809,Z 611.91,A -85,B 0,C 180,E1 11337.717,E2 11337.717} C_VEL
LIN {X 0,Y 380.593,Z 611.91,A -85,B 0,C 180,E1 11344.559,E2 11344.559} C_VEL
LIN {X 0,Y 380.178,Z 611.91,A -85,B 0,C 180,E1 11351.481,E2 11351.481} C_VEL
LIN {X 0,Y 379.908,Z 611.91,A -85,B 0,C 180,E1 11358.587,E2 11358.587} C_VEL
LIN {X 0,Y 379.615,Z 611.91,A -85,B 0,C 180,E1 11366.017,E2 11366.017} C_VEL
LIN {X 0,Y 379.343,Z 611.91,A -85,B 0,C 180,E1 11373.965,E2 11373.965} C_VEL
LIN {X 0,Y 379.196,Z 611.91,A -85,B 0,C 180,E1 11380.656,E2 11380.656} C_VEL
LIN {X 0,Y 379.456,Z 612.353,A -85,B 0,C 180,E1 11386.822,E2 11386.822} C_VEL
LIN {X 0,Y 384.53,Z 622.54,A -85,B 0,C 180,E1 11387.774,E2 11387.774} C_VEL
LIN {X 0,Y 402.838,Z 657.821,A -85,B 0,C 180,E1 11391.026,E2 11391.026} C_VEL
LIN {X 0,Y 410.898,Z 679.941,A -85,B 0,C 180,E1 11392.865,E2 11392.865} C_VEL
LIN {X 0,Y 406.365,Z 715.715,A -85,B 0,C 180,E1 11394.724,E2 11394.724} C_VEL
LIN {X 0,Y 400.721,Z 750.088,A -85,B 0,C 180,E1 11397.424,E2 11397.424} C_VEL
LIN {X 0,Y 394.657,Z 781.834,A -85,B 0,C 180,E1 11401.031,E2 11401.031} C_VEL
LIN {X 0,Y 389.428,Z 807.873,A -85,B 0,C 180,E1 11405.08,E2 11405.08} C_VEL
LIN {X 0,Y 384.98,Z 831.541,A -85,B 0,C 180,E1 11410.185,E2 11410.185} C_VEL
LIN {X 0,Y 382.427,Z 848.937,A -85,B 0,C 180,E1 11415.594,E2 11415.594} C_VEL
LIN {X 0,Y 381.398,Z 860.155,A -85,B 0,C 180,E1 11420.863,E2 11420.863} C_VEL
LIN {X 0,Y 381.075,Z 865.686,A -85,B 0,C 180,E1 11425.442,E2 11425.442} C_VEL
LIN {X 0,Y 381.03,Z 867.442,A -85,B 0,C 180,E1 11430.305,E2 11430.305} C_VEL
LIN {X 0,Y 378.438,Z 866.993,A -85,B 0,C 180,E1 11432.239,E2 11432.239} C_VEL
LIN {X 0,Y 373.323,Z 864.997,A -85,B 0,C 180,E1 11435.142,E2 11435.142} C_VEL
LIN {X 0,Y 373.266,Z 864.665,A -85,B 0,C 180,E1 11435.476,E2 11435.476} C_VEL
LIN {X 0,Y 373.735,Z 856.835,A -85,B 0,C 180,E1 11441.095,E2 11441.095} C_VEL
LIN {X 0,Y 375.286,Z 844.07,A -85,B 0,C 180,E1 11446.404,E2 11446.404} C_VEL
LIN {X 0,Y 378.508,Z 825.368,A -85,B 0,C 180,E1 11451.716,E2 11451.716} C_VEL
LIN {X 0,Y 383.424,Z 801.169,A -85,B 0,C 180,E1 11456.568,E2 11456.568} C_VEL
LIN {X 0,Y 389.161,Z 774.047,A -85,B 0,C 180,E1 11460.55,E2 11460.55} C_VEL
LIN {X 0,Y 395.682,Z 740.679,A -85,B 0,C 180,E1 11464.029,E2 11464.029} C_VEL
LIN {X 0,Y 401.094,Z 708.041,A -85,B 0,C 180,E1 11466.395,E2 11466.395} C_VEL
LIN {X 0,Y 403.842,Z 679.817,A -85,B 0,C 180,E1 11467.89,E2 11467.89} C_VEL
LIN {X 0,Y 390.226,Z 647.099,A -85,B 0,C 180,E1 11470.841,E2 11470.841} C_VEL
LIN {X 0,Y 371.585,Z 613.714,A -85,B 0,C 180,E1 11474.284,E2 11474.284} C_VEL
LIN {X 0,Y 371.342,Z 611.91,A -85,B 0,C 180,E1 11474.556,E2 11474.556} C_VEL
LIN {X 0,Y 371.263,Z 611.91,A -85,B 0,C 180,E1 11480.791,E2 11480.791} C_VEL
LIN {X 0,Y 371.499,Z 611.91,A -85,B 0,C 180,E1 11488.013,E2 11488.013} C_VEL
LIN {X 0,Y 371.659,Z 611.91,A -85,B 0,C 180,E1 11495.965,E2 11495.965} C_VEL
LIN {X 0,Y 372.065,Z 611.91,A -85,B 0,C 180,E1 11503.455,E2 11503.455} C_VEL
LIN {X 0,Y 372.382,Z 611.91,A -85,B 0,C 180,E1 11510.645,E2 11510.645} C_VEL
LIN {X 0,Y 372.785,Z 611.91,A -85,B 0,C 180,E1 11517.677,E2 11517.677} C_VEL
LIN {X 0,Y 372.892,Z 611.91,A -85,B 0,C 180,E1 11522.331,E2 11522.331} C_VEL
LIN {X 0,Y 372.375,Z 611.91,A -85,B 0,C 180,E1 11529.364,E2 11529.364} C_VEL
LIN {X 0,Y 372.072,Z 611.91,A -85,B 0,C 180,E1 11536.553,E2 11536.553} C_VEL
LIN {X 0,Y 371.694,Z 611.91,A -85,B 0,C 180,E1 11544.041,E2 11544.041} C_VEL
LIN {X 0,Y 371.48,Z 611.91,A -85,B 0,C 180,E1 11551.999,E2 11551.999} C_VEL
LIN {X 0,Y 371.296,Z 611.91,A -85,B 0,C 180,E1 11559.215,E2 11559.215} C_VEL
LIN {X 0,Y 371.294,Z 611.91,A -85,B 0,C 180,E1 11566.114,E2 11566.114} C_VEL
LIN {X 0,Y 371.248,Z 611.91,A -85,B 0,C 180,E1 11572.284,E2 11572.284} C_VEL
LIN {X 0,Y 371.48,Z 611.91,A -85,B 0,C 180,E1 11578.864,E2 11578.864} C_VEL
LIN {X 0,Y 371.717,Z 611.91,A -85,B 0,C 180,E1 11585.964,E2 11585.964} C_VEL
LIN {X 0,Y 372.059,Z 611.91,A -85,B 0,C 180,E1 11593.45,E2 11593.45} C_VEL
LIN {X 0,Y 372.379,Z 611.91,A -85,B 0,C 180,E1 11600.64,E2 11600.64} C_VEL
LIN {X 0,Y 372.683,Z 612.85,A -85,B 0,C 180,E1 11605.704,E2 11605.704} C_VEL
LIN {X 0,Y 373.045,Z 613.465,A -85,B 0,C 180,E1 11610,E2 11610} C_VEL
LIN {X 0,Y 372.607,Z 612.055,A -85,B 0,C 180,E1 11614.886,E2 11614.886} C_VEL
LIN {X 0,Y 372.236,Z 611.91,A -85,B 0,C 180,E1 11621.734,E2 11621.734} C_VEL
LIN {X 0,Y 371.943,Z 611.91,A -85,B 0,C 180,E1 11629.005,E2 11629.005} C_VEL
LIN {X 0,Y 371.64,Z 611.91,A -85,B 0,C 180,E1 11636.624,E2 11636.624} C_VEL
LIN {X 0,Y 371.54,Z 611.91,A -85,B 0,C 180,E1 11641.989,E2 11641.989} C_VEL
LIN {X 0,Y 371.298,Z 611.91,A -85,B 0,C 180,E1 11649.212,E2 11649.212} C_VEL
LIN {X 0,Y 371.177,Z 611.91,A -85,B 0,C 180,E1 11656.093,E2 11656.093} C_VEL
LIN {X 0,Y 371.193,Z 611.91,A -85,B 0,C 180,E1 11662.274,E2 11662.274} C_VEL
LIN {X 0,Y 371.477,Z 611.91,A -85,B 0,C 180,E1 11668.861,E2 11668.861} C_VEL
LIN {X 0,Y 371.748,Z 611.91,A -85,B 0,C 180,E1 11675.962,E2 11675.962} C_VEL
LIN {X 0,Y 371.967,Z 611.91,A -85,B 0,C 180,E1 11680.992,E2 11680.992} C_VEL
LIN {X 0,Y 372.129,Z 611.91,A -85,B 0,C 180,E1 11688.258,E2 11688.258} C_VEL
LIN {X 0,Y 372.628,Z 611.91,A -85,B 0,C 180,E1 11695.335,E2 11695.335} C_VEL
LIN {X 0,Y 372.941,Z 611.91,A -85,B 0,C 180,E1 11699.996,E2 11699.996} C_VEL
LIN {X 0,Y 372.501,Z 611.91,A -85,B 0,C 180,E1 11706.999,E2 11706.999} C_VEL
LIN {X 0,Y 372.142,Z 611.91,A -85,B 0,C 180,E1 11714.124,E2 11714.124} C_VEL
LIN {X 0,Y 371.83,Z 611.91,A -85,B 0,C 180,E1 11721.493,E2 11721.493} C_VEL
LIN {X 0,Y 371.623,Z 611.91,A -85,B 0,C 180,E1 11726.62,E2 11726.62} C_VEL
LIN {X 0,Y 371.461,Z 611.91,A -85,B 0,C 180,E1 11731.99,E2 11731.99} C_VEL
LIN {X 0,Y 371.25,Z 611.91,A -85,B 0,C 180,E1 11739.207,E2 11739.207} C_VEL
LIN {X 0,Y 371.39,Z 612.12,A -85,B 0,C 180,E1 11745.645,E2 11745.645} C_VEL
LIN {X 0,Y 374.084,Z 617.811,A -85,B 0,C 180,E1 11746.192,E2 11746.192} C_VEL
LIN {X 0,Y 394.122,Z 655.131,A -85,B 0,C 180,E1 11749.899,E2 11749.899} C_VEL
LIN {X 0,Y 404.254,Z 680.997,A -85,B 0,C 180,E1 11752.212,E2 11752.212} C_VEL
LIN {X 0,Y 399.537,Z 717.675,A -85,B 0,C 180,E1 11754.211,E2 11754.211} C_VEL
LIN {X 0,Y 393.699,Z 751.265,A -85,B 0,C 180,E1 11756.934,E2 11756.934} C_VEL
LIN {X 0,Y 387.159,Z 783.723,A -85,B 0,C 180,E1 11760.736,E2 11760.736} C_VEL
LIN {X 0,Y 381.562,Z 810.111,A -85,B 0,C 180,E1 11765.047,E2 11765.047} C_VEL
LIN {X 0,Y 377.166,Z 832.46,A -85,B 0,C 180,E1 11770.065,E2 11770.065} C_VEL
LIN {X 0,Y 374.614,Z 848.907,A -85,B 0,C 180,E1 11775.368,E2 11775.368} C_VEL
LIN {X 0,Y 373.512,Z 859.919,A -85,B 0,C 180,E1 11780.669,E2 11780.669} C_VEL
LIN {X 0,Y 373.202,Z 865.452,A -85,B 0,C 180,E1 11785.346,E2 11785.346} C_VEL
LIN {X 0,Y 373.154,Z 867.215,A -85,B 0,C 180,E1 11790.283,E2 11790.283} C_VEL
LIN {X 0,Y 373.266,Z 864.665,A -85,B 0,C 180,E1 11795.476,E2 11795.476} C_VEL
LIN {X 0,Y 370.905,Z 862.565,A -85,B 0,C 180,E1 11797.434,E2 11797.434} C_VEL
LIN {X 0,Y 365.835,Z 858.286,A -85,B 0,C 180,E1 11800.355,E2 11800.355} C_VEL
LIN {X 0,Y 365.79,Z 857.705,A -85,B 0,C 180,E1 11800.689,E2 11800.689} C_VEL
LIN {X 0,Y 367.304,Z 845.606,A -85,B 0,C 180,E1 11806.155,E2 11806.155} C_VEL
LIN {X 0,Y 370.73,Z 826.304,A -85,B 0,C 180,E1 11811.88,E2 11811.88} C_VEL
LIN {X 0,Y 375.758,Z 802.862,A -85,B 0,C 180,E1 11816.784,E2 11816.784} C_VEL
LIN {X 0,Y 381.983,Z 774.968,A -85,B 0,C 180,E1 11821.016,E2 11821.016} C_VEL
LIN {X 0,Y 388.447,Z 743.499,A -85,B 0,C 180,E1 11824.414,E2 11824.414} C_VEL
LIN {X 0,Y 394.373,Z 710.155,A -85,B 0,C 180,E1 11826.946,E2 11826.946} C_VEL
LIN {X 0,Y 397.584,Z 682.98,A -85,B 0,C 180,E1 11828.418,E2 11828.418} C_VEL
LIN {X 0,Y 384.473,Z 650.866,A -85,B 0,C 180,E1 11831.466,E2 11831.466} C_VEL
LIN {X 0,Y 365.748,Z 617.534,A -85,B 0,C 180,E1 11835.072,E2 11835.072} C_VEL
LIN {X 0,Y 363.377,Z 611.91,A -85,B 0,C 180,E1 11835.768,E2 11835.768} C_VEL
LIN {X 0,Y 363.368,Z 611.91,A -85,B 0,C 180,E1 11842.343,E2 11842.343} C_VEL
LIN {X 0,Y 363.625,Z 611.91,A -85,B 0,C 180,E1 11850.029,E2 11850.029} C_VEL
LIN {X 0,Y 363.799,Z 611.91,A -85,B 0,C 180,E1 11858.008,E2 11858.008} C_VEL
LIN {X 0,Y 364.19,Z 611.91,A -85,B 0,C 180,E1 11865.561,E2 11865.561} C_VEL
LIN {X 0,Y 364.579,Z 611.91,A -85,B 0,C 180,E1 11872.848,E2 11872.848} C_VEL
LIN {X 0,Y 364.975,Z 611.91,A -85,B 0,C 180,E1 11880.004,E2 11880.004} C_VEL
LIN {X 0,Y 364.669,Z 611.91,A -85,B 0,C 180,E1 11887.159,E2 11887.159} C_VEL
LIN {X 0,Y 364.201,Z 611.91,A -85,B 0,C 180,E1 11894.448,E2 11894.448} C_VEL
LIN {X 0,Y 363.831,Z 611.91,A -85,B 0,C 180,E1 11901.999,E2 11901.999} C_VEL
LIN {X 0,Y 363.597,Z 611.91,A -85,B 0,C 180,E1 11909.983,E2 11909.983} C_VEL
LIN {X 0,Y 363.394,Z 611.91,A -85,B 0,C 180,E1 11917.663,E2 11917.663} C_VEL
LIN {X 0,Y 363.337,Z 611.91,A -85,B 0,C 180,E1 11925.109,E2 11925.109} C_VEL
LIN {X 0,Y 363.36,Z 611.91,A -85,B 0,C 180,E1 11932.348,E2 11932.348} C_VEL
LIN {X 0,Y 363.592,Z 611.91,A -85,B 0,C 180,E1 11940.02,E2 11940.02} C_VEL
LIN {X 0,Y 363.84,Z 611.91,A -85,B 0,C 180,E1 11948.005,E2 11948.005} C_VEL
LIN {X 0,Y 364.014,Z 612.637,A -85,B 0,C 180,E1 11950.129,E2 11950.129} C_VEL
LIN {X 0,Y 365.756,Z 616.795,A -85,B 0,C 180,E1 11952.845,E2 11952.845} C_VEL
LIN {X 0,Y 369.301,Z 619.256,A -85,B 0,C 180,E1 11958.711,E2 11958.711} C_VEL
LIN {X 0,Y 371.596,Z 620.089,A -85,B 0,C 180,E1 11965.033,E2 11965.033} C_VEL
LIN {X 0,Y 372.083,Z 621.305,A -85,B 0,C 180,E1 11970,E2 11970} C_VEL
LIN {X 0,Y 371.617,Z 619.925,A -85,B 0,C 180,E1 11974.967,E2 11974.967} C_VEL
LIN {X 0,Y 369.301,Z 619.252,A -85,B 0,C 180,E1 11981.289,E2 11981.289} C_VEL
LIN {X 0,Y 365.872,Z 616.877,A -85,B 0,C 180,E1 11986.994,E2 11986.994} C_VEL
LIN {X 0,Y 364.018,Z 612.603,A -85,B 0,C 180,E1 11989.871,E2 11989.871} C_VEL
LIN {X 0,Y 363.649,Z 611.91,A -85,B 0,C 180,E1 11997.257,E2 11997.257} C_VEL
LIN {X 0,Y 363.478,Z 611.91,A -85,B 0,C 180,E1 12003.578,E2 12003.578} C_VEL
LIN {X 0,Y 363.402,Z 611.91,A -85,B 0,C 180,E1 12008.679,E2 12008.679} C_VEL
LIN {X 0,Y 363.232,Z 611.91,A -85,B 0,C 180,E1 12015.122,E2 12015.122} C_VEL
LIN {X 0,Y 363.309,Z 611.91,A -85,B 0,C 180,E1 12022.355,E2 12022.355} C_VEL
LIN {X 0,Y 363.597,Z 611.91,A -85,B 0,C 180,E1 12030.017,E2 12030.017} C_VEL
LIN {X 0,Y 363.89,Z 611.91,A -85,B 0,C 180,E1 12038.005,E2 12038.005} C_VEL
LIN {X 0,Y 364.116,Z 611.91,A -85,B 0,C 180,E1 12045.549,E2 12045.549} C_VEL
LIN {X 0,Y 364.662,Z 611.91,A -85,B 0,C 180,E1 12052.841,E2 12052.841} C_VEL
LIN {X 0,Y 365.038,Z 611.91,A -85,B 0,C 180,E1 12059.996,E2 12059.996} C_VEL
LIN {X 0,Y 364.579,Z 611.91,A -85,B 0,C 180,E1 12067.152,E2 12067.152} C_VEL
LIN {X 0,Y 364.195,Z 611.91,A -85,B 0,C 180,E1 12074.439,E2 12074.439} C_VEL
LIN {X 0,Y 363.846,Z 611.91,A -85,B 0,C 180,E1 12081.989,E2 12081.989} C_VEL
LIN {X 0,Y 363.586,Z 611.91,A -85,B 0,C 180,E1 12089.974,E2 12089.974} C_VEL
LIN {X 0,Y 363.344,Z 611.91,A -85,B 0,C 180,E1 12097.653,E2 12097.653} C_VEL
LIN {X 0,Y 363.381,Z 611.91,A -85,B 0,C 180,E1 12104.374,E2 12104.374} C_VEL
LIN {X 0,Y 366.06,Z 617.811,A -85,B 0,C 180,E1 12104.984,E2 12104.984} C_VEL
LIN {X 0,Y 386.193,Z 654.373,A -85,B 0,C 180,E1 12108.882,E2 12108.882} C_VEL
LIN {X 0,Y 397.829,Z 684.017,A -85,B 0,C 180,E1 12111.673,E2 12111.673} C_VEL
LIN {X 0,Y 392.287,Z 722.317,A -85,B 0,C 180,E1 12113.859,E2 12113.859} C_VEL
LIN {X 0,Y 386.137,Z 755.074,A -85,B 0,C 180,E1 12116.705,E2 12116.705} C_VEL
LIN {X 0,Y 379.668,Z 785.589,A -85,B 0,C 180,E1 12120.429,E2 12120.429} C_VEL
LIN {X 0,Y 373.565,Z 812.96,A -85,B 0,C 180,E1 12125.134,E2 12125.134} C_VEL
LIN {X 0,Y 369.347,Z 833.312,A -85,B 0,C 180,E1 12129.953,E2 12129.953} C_VEL
LIN {X 0,Y 366.618,Z 850.189,A -85,B 0,C 180,E1 12135.653,E2 12135.653} C_VEL
LIN {X 0,Y 365.648,Z 859.683,A -85,B 0,C 180,E1 12140.466,E2 12140.466} C_VEL
LIN {X 0,Y 365.307,Z 865.218,A -85,B 0,C 180,E1 12145.245,E2 12145.245} C_VEL
LIN {X 0,Y 365.294,Z 867.037,A -85,B 0,C 180,E1 12150,E2 12150} C_VEL
LIN {X 0,Y 365.323,Z 864.536,A -85,B 0,C 180,E1 12155.481,E2 12155.481} C_VEL
LIN {X 0,Y 365.79,Z 857.705,A -85,B 0,C 180,E1 12160.689,E2 12160.689} C_VEL
LIN {X 0,Y 364.76,Z 855.367,A -85,B 0,C 180,E1 12162.001,E2 12162.001} C_VEL
LIN {X 0,Y 359.217,Z 847.776,A -85,B 0,C 180,E1 12165.547,E2 12165.547} C_VEL
LIN {X 0,Y 359.264,Z 846.967,A -85,B 0,C 180,E1 12165.875,E2 12165.875} C_VEL
LIN {X 0,Y 362.472,Z 829.594,A -85,B 0,C 180,E1 12171.438,E2 12171.438} C_VEL
LIN {X 0,Y 367.643,Z 806.705,A -85,B 0,C 180,E1 12176.607,E2 12176.607} C_VEL
LIN {X 0,Y 374.062,Z 778.987,A -85,B 0,C 180,E1 12181.069,E2 12181.069} C_VEL
LIN {X 0,Y 380.912,Z 748.443,A -85,B 0,C 180,E1 12184.606,E2 12184.606} C_VEL
LIN {X 0,Y 387.473,Z 713.004,A -85,B 0,C 180,E1 12187.453,E2 12187.453} C_VEL
LIN {X 0,Y 390.983,Z 685.229,A -85,B 0,C 180,E1 12189.032,E2 12189.032} C_VEL
LIN {X 0,Y 378.43,Z 653.946,A -85,B 0,C 180,E1 12192.157,E2 12192.157} C_VEL
LIN {X 0,Y 360.798,Z 622.534,A -85,B 0,C 180,E1 12195.72,E2 12195.72} C_VEL
LIN {X 0,Y 355.56,Z 613.367,A -85,B 0,C 180,E1 12196.85,E2 12196.85} C_VEL
LIN {X 0,Y 355.415,Z 611.91,A -85,B 0,C 180,E1 12197.04,E2 12197.04} C_VEL
LIN {X 0,Y 355.47,Z 611.91,A -85,B 0,C 180,E1 12204.025,E2 12204.025} C_VEL
LIN {X 0,Y 355.72,Z 611.91,A -85,B 0,C 180,E1 12212.089,E2 12212.089} C_VEL
LIN {X 0,Y 355.999,Z 611.91,A -85,B 0,C 180,E1 12220.114,E2 12220.114} C_VEL
LIN {X 0,Y 356.382,Z 611.91,A -85,B 0,C 180,E1 12227.741,E2 12227.741} C_VEL
LIN {X 0,Y 356.821,Z 611.91,A -85,B 0,C 180,E1 12235.136,E2 12235.136} C_VEL
LIN {X 0,Y 357.087,Z 611.91,A -85,B 0,C 180,E1 12242.434,E2 12242.434} C_VEL
LIN {X 0,Y 356.495,Z 611.91,A -85,B 0,C 180,E1 12249.785,E2 12249.785} C_VEL
LIN {X 0,Y 356.193,Z 611.91,A -85,B 0,C 180,E1 12257.314,E2 12257.314} C_VEL
LIN {X 0,Y 355.75,Z 611.91,A -85,B 0,C 180,E1 12265.192,E2 12265.192} C_VEL
LIN {X 0,Y 355.508,Z 611.91,A -85,B 0,C 180,E1 12271.595,E2 12271.595} C_VEL
LIN {X 0,Y 355.454,Z 611.91,A -85,B 0,C 180,E1 12276.611,E2 12276.611} C_VEL
LIN {X 0,Y 355.33,Z 611.91,A -85,B 0,C 180,E1 12283.584,E2 12283.584} C_VEL
